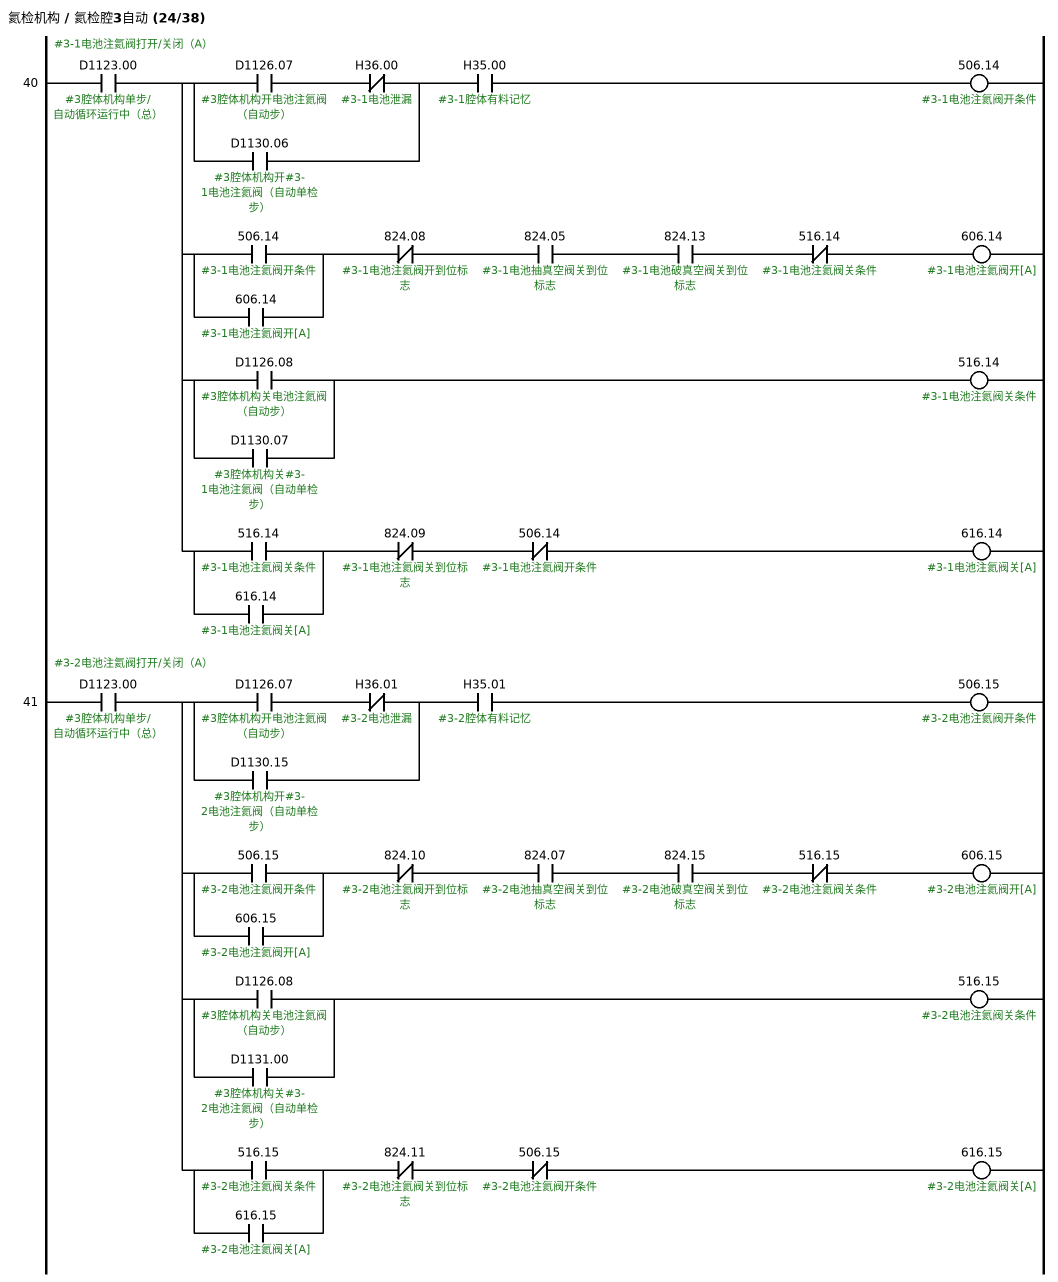
; [picture p312: 氦检机构 / 氦检腔3自动, rungs 40-41]
; rung 40: #3-1电池注氦阀打开/关闭（A）
LD D1123.00  ; #3腔体机构单步/自动循环运行中（总）
OUT TR0
LD D1126.07  ; #3腔体机构开电池注氦阀（自动步）
ANDNOT H36.00  ; #3-1电池泄漏
OR D1130.06  ; #3腔体机构开#3-1电池注氦阀（自动单检步）
ANDLD
AND H35.00  ; #3-1腔体有料记忆
OUT 506.14  ; #3-1电池注氦阀开条件
LD TR0
LD 506.14  ; #3-1电池注氦阀开条件
OR 606.14  ; #3-1电池注氦阀开[A]
ANDLD
ANDNOT 824.08  ; #3-1电池注氦阀开到位标志
AND 824.05  ; #3-1电池抽真空阀关到位标志
AND 824.13  ; #3-1电池破真空阀关到位标志
ANDNOT 516.14  ; #3-1电池注氦阀关条件
OUT 606.14  ; #3-1电池注氦阀开[A]
LD TR0
LD D1126.08  ; #3腔体机构关电池注氦阀（自动步）
OR D1130.07  ; #3腔体机构关#3-1电池注氦阀（自动单检步）
ANDLD
OUT 516.14  ; #3-1电池注氦阀关条件
LD TR0
LD 516.14  ; #3-1电池注氦阀关条件
OR 616.14  ; #3-1电池注氦阀关[A]
ANDLD
ANDNOT 824.09  ; #3-1电池注氦阀关到位标志
ANDNOT 506.14  ; #3-1电池注氦阀开条件
OUT 616.14  ; #3-1电池注氦阀关[A]
; rung 41: #3-2电池注氦阀打开/关闭（A）
LD D1123.00  ; #3腔体机构单步/自动循环运行中（总）
OUT TR0
LD D1126.07  ; #3腔体机构开电池注氦阀（自动步）
ANDNOT H36.01  ; #3-2电池泄漏
OR D1130.15  ; #3腔体机构开#3-2电池注氦阀（自动单检步）
ANDLD
AND H35.01  ; #3-2腔体有料记忆
OUT 506.15  ; #3-2电池注氦阀开条件
LD TR0
LD 506.15  ; #3-2电池注氦阀开条件
OR 606.15  ; #3-2电池注氦阀开[A]
ANDLD
ANDNOT 824.10  ; #3-2电池注氦阀开到位标志
AND 824.07  ; #3-2电池抽真空阀关到位标志
AND 824.15  ; #3-2电池破真空阀关到位标志
ANDNOT 516.15  ; #3-2电池注氦阀关条件
OUT 606.15  ; #3-2电池注氦阀开[A]
LD TR0
LD D1126.08  ; #3腔体机构关电池注氦阀（自动步）
OR D1131.00  ; #3腔体机构关#3-2电池注氦阀（自动单检步）
ANDLD
OUT 516.15  ; #3-2电池注氦阀关条件
LD TR0
LD 516.15  ; #3-2电池注氦阀关条件
OR 616.15  ; #3-2电池注氦阀关[A]
ANDLD
ANDNOT 824.11  ; #3-2电池注氦阀关到位标志
ANDNOT 506.15  ; #3-2电池注氦阀开条件
OUT 616.15  ; #3-2电池注氦阀关[A]

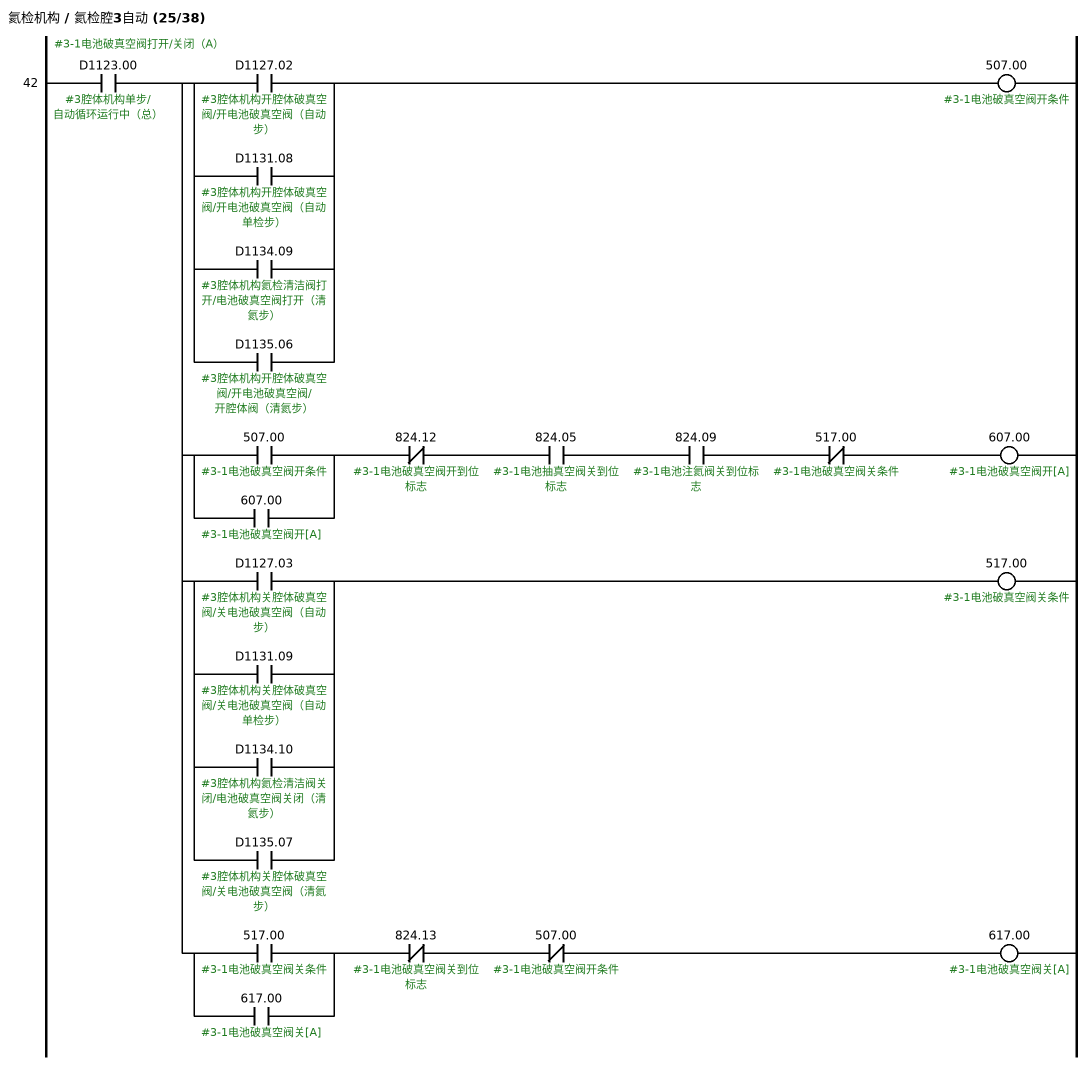
; rung 42: #3-1电池破真空阀打开/关闭（A）
LD D1123.00  ; #3腔体机构单步/自动循环运行中（总）
OUT TR0
LD D1127.02  ; #3腔体机构开腔体破真空阀/开电池破真空阀（自动步）
OR D1131.08  ; #3腔体机构开腔体破真空阀/开电池破真空阀（自动单检步）
OR D1134.09  ; #3腔体机构氦检清洁阀打开/电池破真空阀打开（清氦步）
OR D1135.06  ; #3腔体机构开腔体破真空阀/开电池破真空阀/开腔体阀（清氦步）
ANDLD
OUT 507.00  ; #3-1电池破真空阀开条件
LD TR0
LD 507.00  ; #3-1电池破真空阀开条件
OR 607.00  ; #3-1电池破真空阀开[A]
ANDLD
ANDNOT 824.12  ; #3-1电池破真空阀开到位标志
AND 824.05  ; #3-1电池抽真空阀关到位标志
AND 824.09  ; #3-1电池注氦阀关到位标志
ANDNOT 517.00  ; #3-1电池破真空阀关条件
OUT 607.00  ; #3-1电池破真空阀开[A]
LD TR0
LD D1127.03  ; #3腔体机构关腔体破真空阀/关电池破真空阀（自动步）
OR D1131.09  ; #3腔体机构关腔体破真空阀/关电池破真空阀（自动单检步）
OR D1134.10  ; #3腔体机构氦检清洁阀关闭/电池破真空阀关闭（清氦步）
OR D1135.07  ; #3腔体机构关腔体破真空阀/关电池破真空阀（清氦步）
ANDLD
OUT 517.00  ; #3-1电池破真空阀关条件
LD TR0
LD 517.00  ; #3-1电池破真空阀关条件
OR 617.00  ; #3-1电池破真空阀关[A]
ANDLD
ANDNOT 824.13  ; #3-1电池破真空阀关到位标志
ANDNOT 507.00  ; #3-1电池破真空阀开条件
OUT 617.00  ; #3-1电池破真空阀关[A]

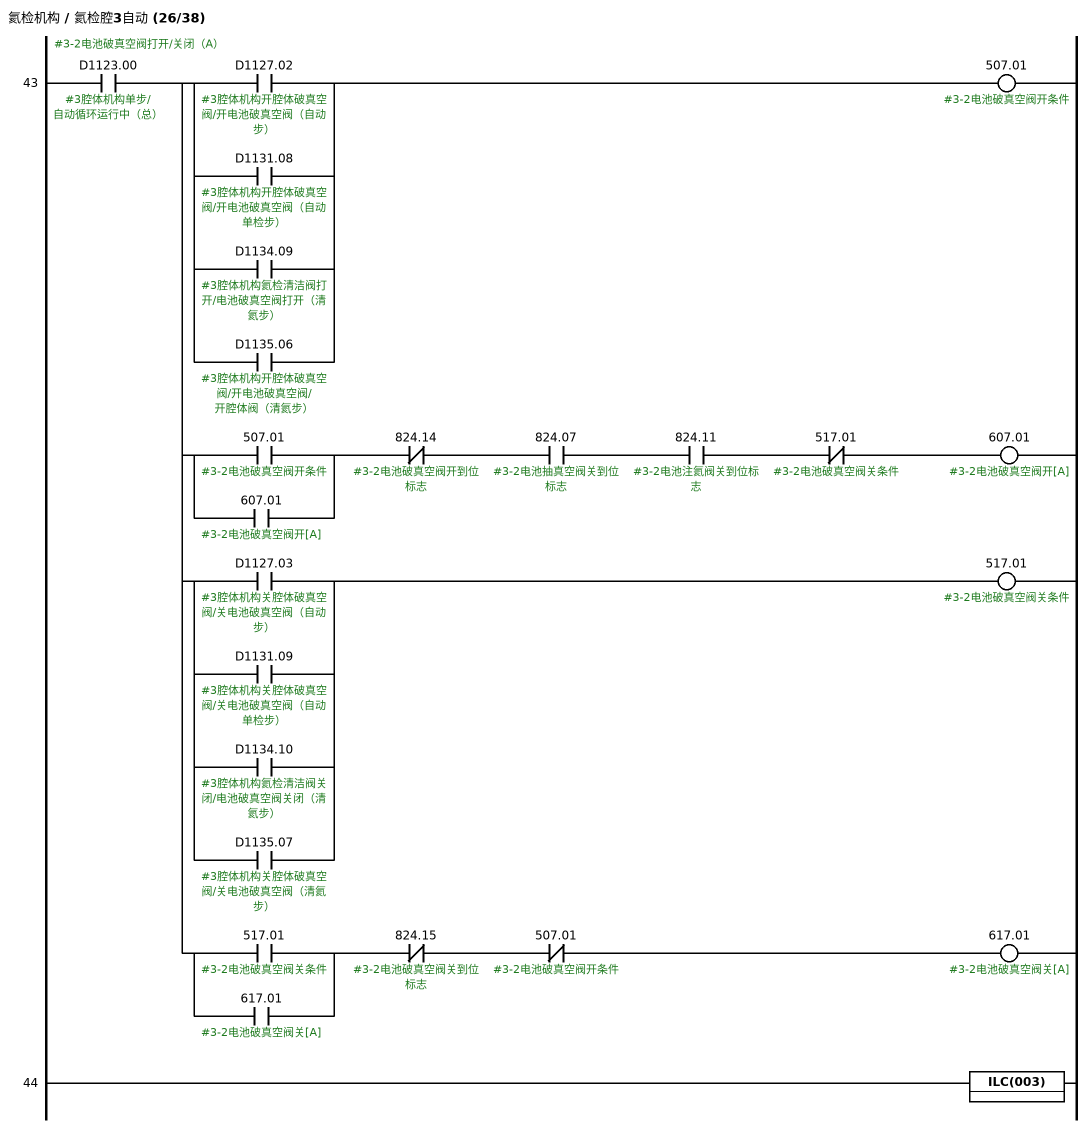
; rung 43: #3-2电池破真空阀打开/关闭（A）
LD D1123.00  ; #3腔体机构单步/自动循环运行中（总）
OUT TR0
LD D1127.02  ; #3腔体机构开腔体破真空阀/开电池破真空阀（自动步）
OR D1131.08  ; #3腔体机构开腔体破真空阀/开电池破真空阀（自动单检步）
OR D1134.09  ; #3腔体机构氦检清洁阀打开/电池破真空阀打开（清氦步）
OR D1135.06  ; #3腔体机构开腔体破真空阀/开电池破真空阀/开腔体阀（清氦步）
ANDLD
OUT 507.01  ; #3-2电池破真空阀开条件
LD TR0
LD 507.01  ; #3-2电池破真空阀开条件
OR 607.01  ; #3-2电池破真空阀开[A]
ANDLD
ANDNOT 824.14  ; #3-2电池破真空阀开到位标志
AND 824.07  ; #3-2电池抽真空阀关到位标志
AND 824.11  ; #3-2电池注氦阀关到位标志
ANDNOT 517.01  ; #3-2电池破真空阀关条件
OUT 607.01  ; #3-2电池破真空阀开[A]
LD TR0
LD D1127.03  ; #3腔体机构关腔体破真空阀/关电池破真空阀（自动步）
OR D1131.09  ; #3腔体机构关腔体破真空阀/关电池破真空阀（自动单检步）
OR D1134.10  ; #3腔体机构氦检清洁阀关闭/电池破真空阀关闭（清氦步）
OR D1135.07  ; #3腔体机构关腔体破真空阀/关电池破真空阀（清氦步）
ANDLD
OUT 517.01  ; #3-2电池破真空阀关条件
LD TR0
LD 517.01  ; #3-2电池破真空阀关条件
OR 617.01  ; #3-2电池破真空阀关[A]
ANDLD
ANDNOT 824.15  ; #3-2电池破真空阀关到位标志
ANDNOT 507.01  ; #3-2电池破真空阀开条件
OUT 617.01  ; #3-2电池破真空阀关[A]
; rung 44
ILC(003)

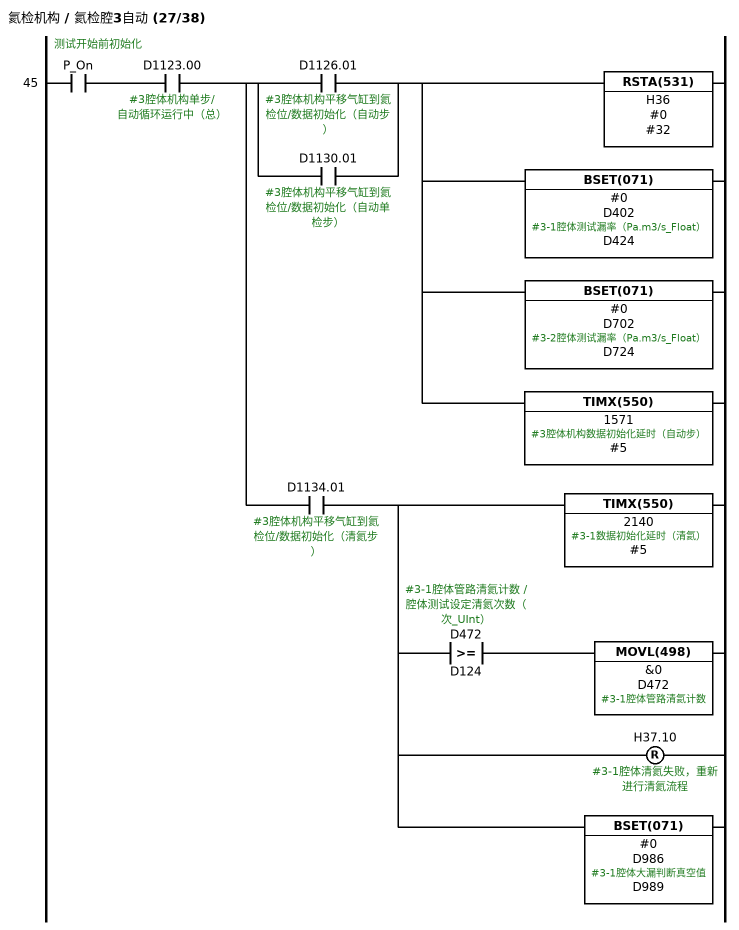
; rung 45: 测试开始前初始化
LD P_On
AND D1123.00  ; #3腔体机构单步/自动循环运行中（总）
OUT TR0
LD D1126.01  ; #3腔体机构平移气缸到氦检位/数据初始化（自动步）
OR D1130.01  ; #3腔体机构平移气缸到氦检位/数据初始化（自动单检步）
ANDLD
RSTA(531) H36 #0 #32
BSET(071) #0 D402 D424  ; #3-1腔体测试漏率（Pa.m3/s_Float）
BSET(071) #0 D702 D724  ; #3-2腔体测试漏率（Pa.m3/s_Float）
TIMX(550) 1571 #5  ; #3腔体机构数据初始化延时（自动步）
LD TR0
AND D1134.01  ; #3腔体机构平移气缸到氦检位/数据初始化（清氦步）
OUT TR0
TIMX(550) 2140 #5  ; #3-1数据初始化延时（清氦）
AND>=(325) D472 D124  ; #3-1腔体管路清氦计数, 腔体测试设定清氦次数（次_UInt）
MOVL(498) &0 D472  ; #3-1腔体管路清氦计数
LD TR0
RSET H37.10  ; #3-1腔体清氦失败，重新进行清氦流程
BSET(071) #0 D986 D989  ; #3-1腔体大漏判断真空值

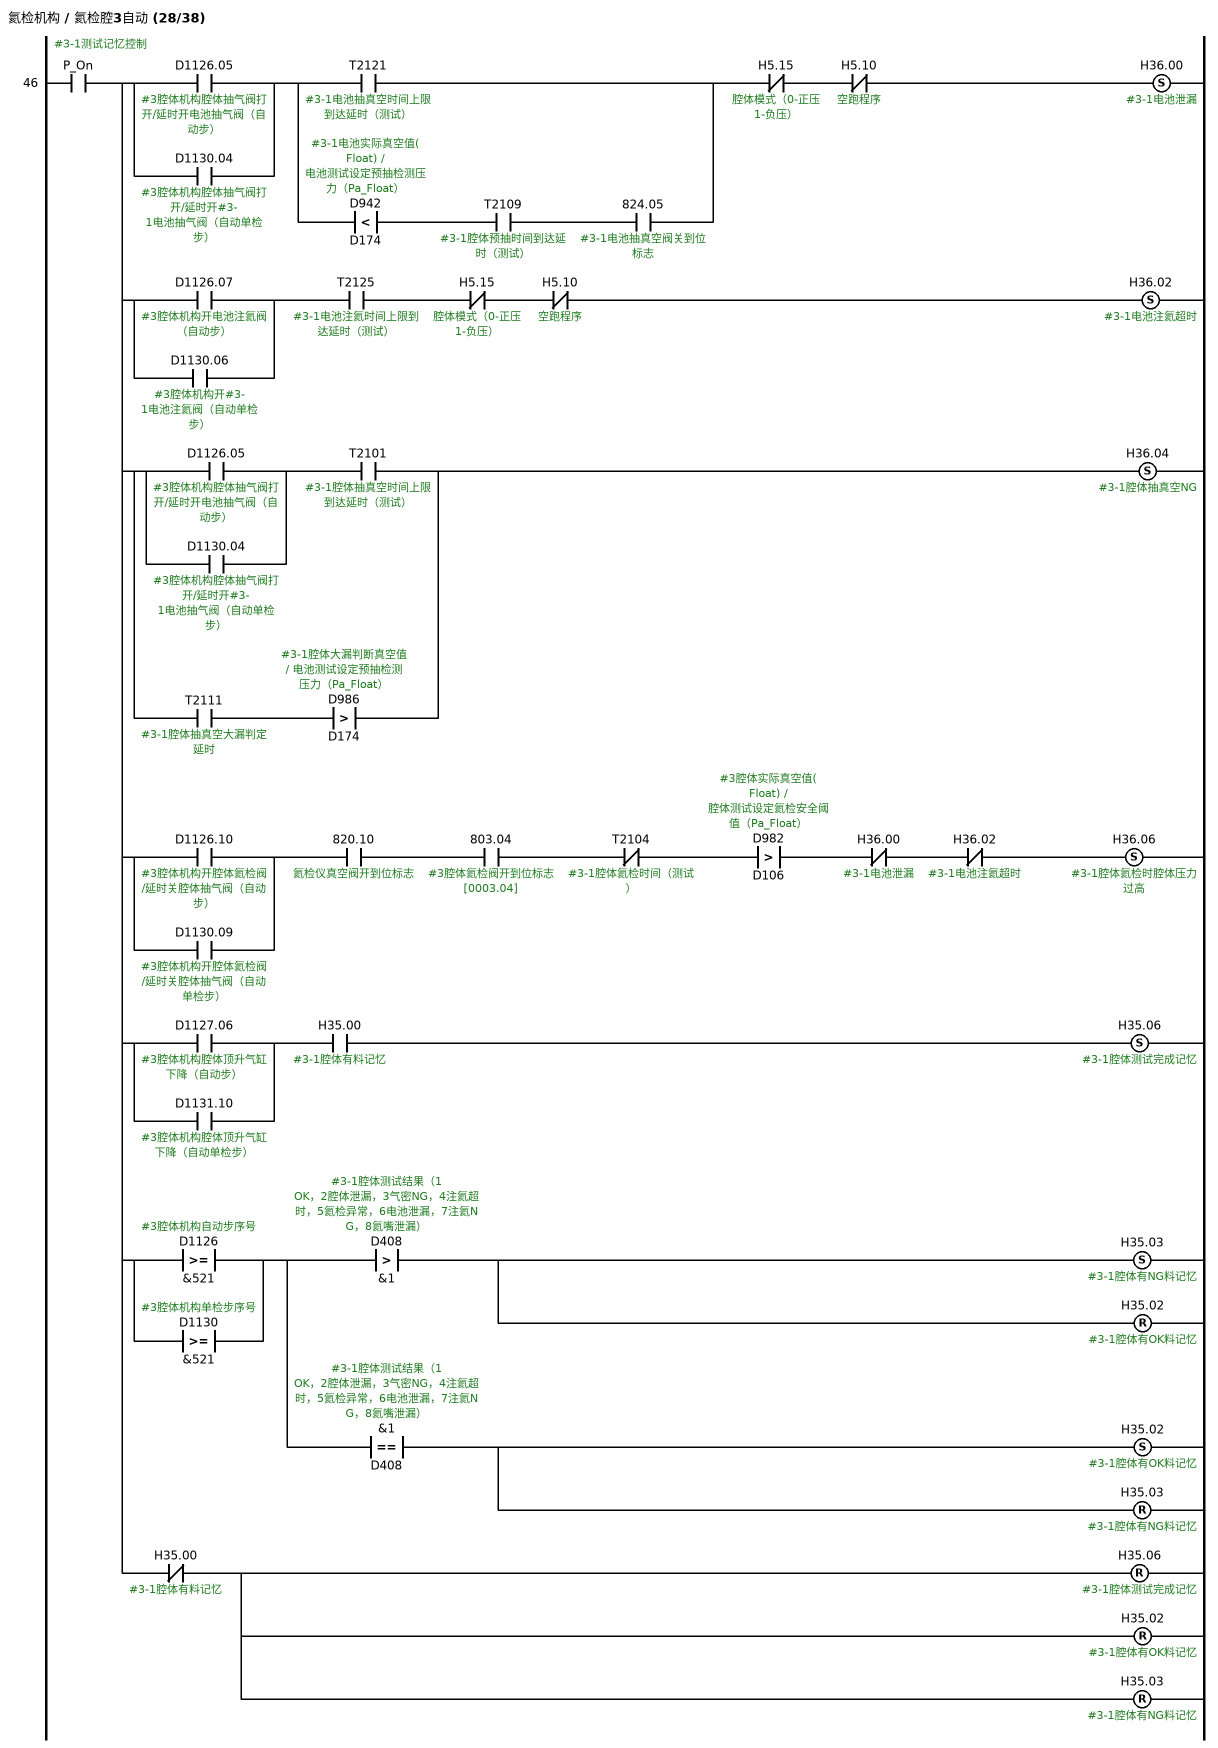
; rung 46: #3-1测试记忆控制
LD P_On
OUT TR0
LD D1126.05  ; #3腔体机构腔体抽气阀打开/延时开电池抽气阀（自动步）
OR D1130.04  ; #3腔体机构腔体抽气阀打开/延时开#3-1电池抽气阀（自动单检步）
ANDLD
LD T2121  ; #3-1电池抽真空时间上限到达延时（测试）
LD<F(331) D942 D174  ; #3-1电池实际真空值(Float), 电池测试设定预抽检测压力（Pa_Float）
AND T2109  ; #3-1腔体预抽时间到达延时（测试）
AND 824.05  ; #3-1电池抽真空阀关到位标志
ORLD
ANDLD
ANDNOT H5.15  ; 腔体模式（0-正压 1-负压）
ANDNOT H5.10  ; 空跑程序
SET H36.00  ; #3-1电池泄漏
LD TR0
LD D1126.07  ; #3腔体机构开电池注氦阀（自动步）
OR D1130.06  ; #3腔体机构开#3-1电池注氦阀（自动单检步）
ANDLD
AND T2125  ; #3-1电池注氦时间上限到达延时（测试）
ANDNOT H5.15  ; 腔体模式（0-正压 1-负压）
ANDNOT H5.10  ; 空跑程序
SET H36.02  ; #3-1电池注氦超时
LD TR0
LD D1126.05  ; #3腔体机构腔体抽气阀打开/延时开电池抽气阀（自动步）
OR D1130.04  ; #3腔体机构腔体抽气阀打开/延时开#3-1电池抽气阀（自动单检步）
AND T2101  ; #3-1腔体抽真空时间上限到达延时（测试）
LD T2111  ; #3-1腔体抽真空大漏判定延时
AND>F(333) D986 D174  ; #3-1腔体大漏判断真空值, 电池测试设定预抽检测压力（Pa_Float）
ORLD
ANDLD
SET H36.04  ; #3-1腔体抽真空NG
LD TR0
LD D1126.10  ; #3腔体机构开腔体氦检阀/延时关腔体抽气阀（自动步）
OR D1130.09  ; #3腔体机构开腔体氦检阀/延时关腔体抽气阀（自动单检步）
ANDLD
AND 820.10  ; 氦检仪真空阀开到位标志
AND 803.04  ; #3腔体氦检阀开到位标志[0003.04]
ANDNOT T2104  ; #3-1腔体氦检时间（测试）
AND>F(333) D982 D106  ; #3腔体实际真空值(Float), 腔体测试设定氦检安全阈值（Pa_Float）
ANDNOT H36.00  ; #3-1电池泄漏
ANDNOT H36.02  ; #3-1电池注氦超时
SET H36.06  ; #3-1腔体氦检时腔体压力过高
LD TR0
LD D1127.06  ; #3腔体机构腔体顶升气缸下降（自动步）
OR D1131.10  ; #3腔体机构腔体顶升气缸下降（自动单检步）
ANDLD
AND H35.00  ; #3-1腔体有料记忆
SET H35.06  ; #3-1腔体测试完成记忆
LD TR0
LD>=L(326) D1126 &521  ; #3腔体机构自动步序号
OR>=L(326) D1130 &521  ; #3腔体机构单检步序号
ANDLD
OUT TR1
AND>(320) D408 &1  ; #3-1腔体测试结果（1 OK，2腔体泄漏，3气密NG，4注氦超时，5氦检异常，6电池泄漏，7注氦NG，8氦嘴泄漏）
SET H35.03  ; #3-1腔体有NG料记忆
RSET H35.02  ; #3-1腔体有OK料记忆
LD TR1
AND=(300) &1 D408  ; #3-1腔体测试结果（1 OK，2腔体泄漏，3气密NG，4注氦超时，5氦检异常，6电池泄漏，7注氦NG，8氦嘴泄漏）
SET H35.02  ; #3-1腔体有OK料记忆
RSET H35.03  ; #3-1腔体有NG料记忆
LD TR0
ANDNOT H35.00  ; #3-1腔体有料记忆
RSET H35.06  ; #3-1腔体测试完成记忆
RSET H35.02  ; #3-1腔体有OK料记忆
RSET H35.03  ; #3-1腔体有NG料记忆

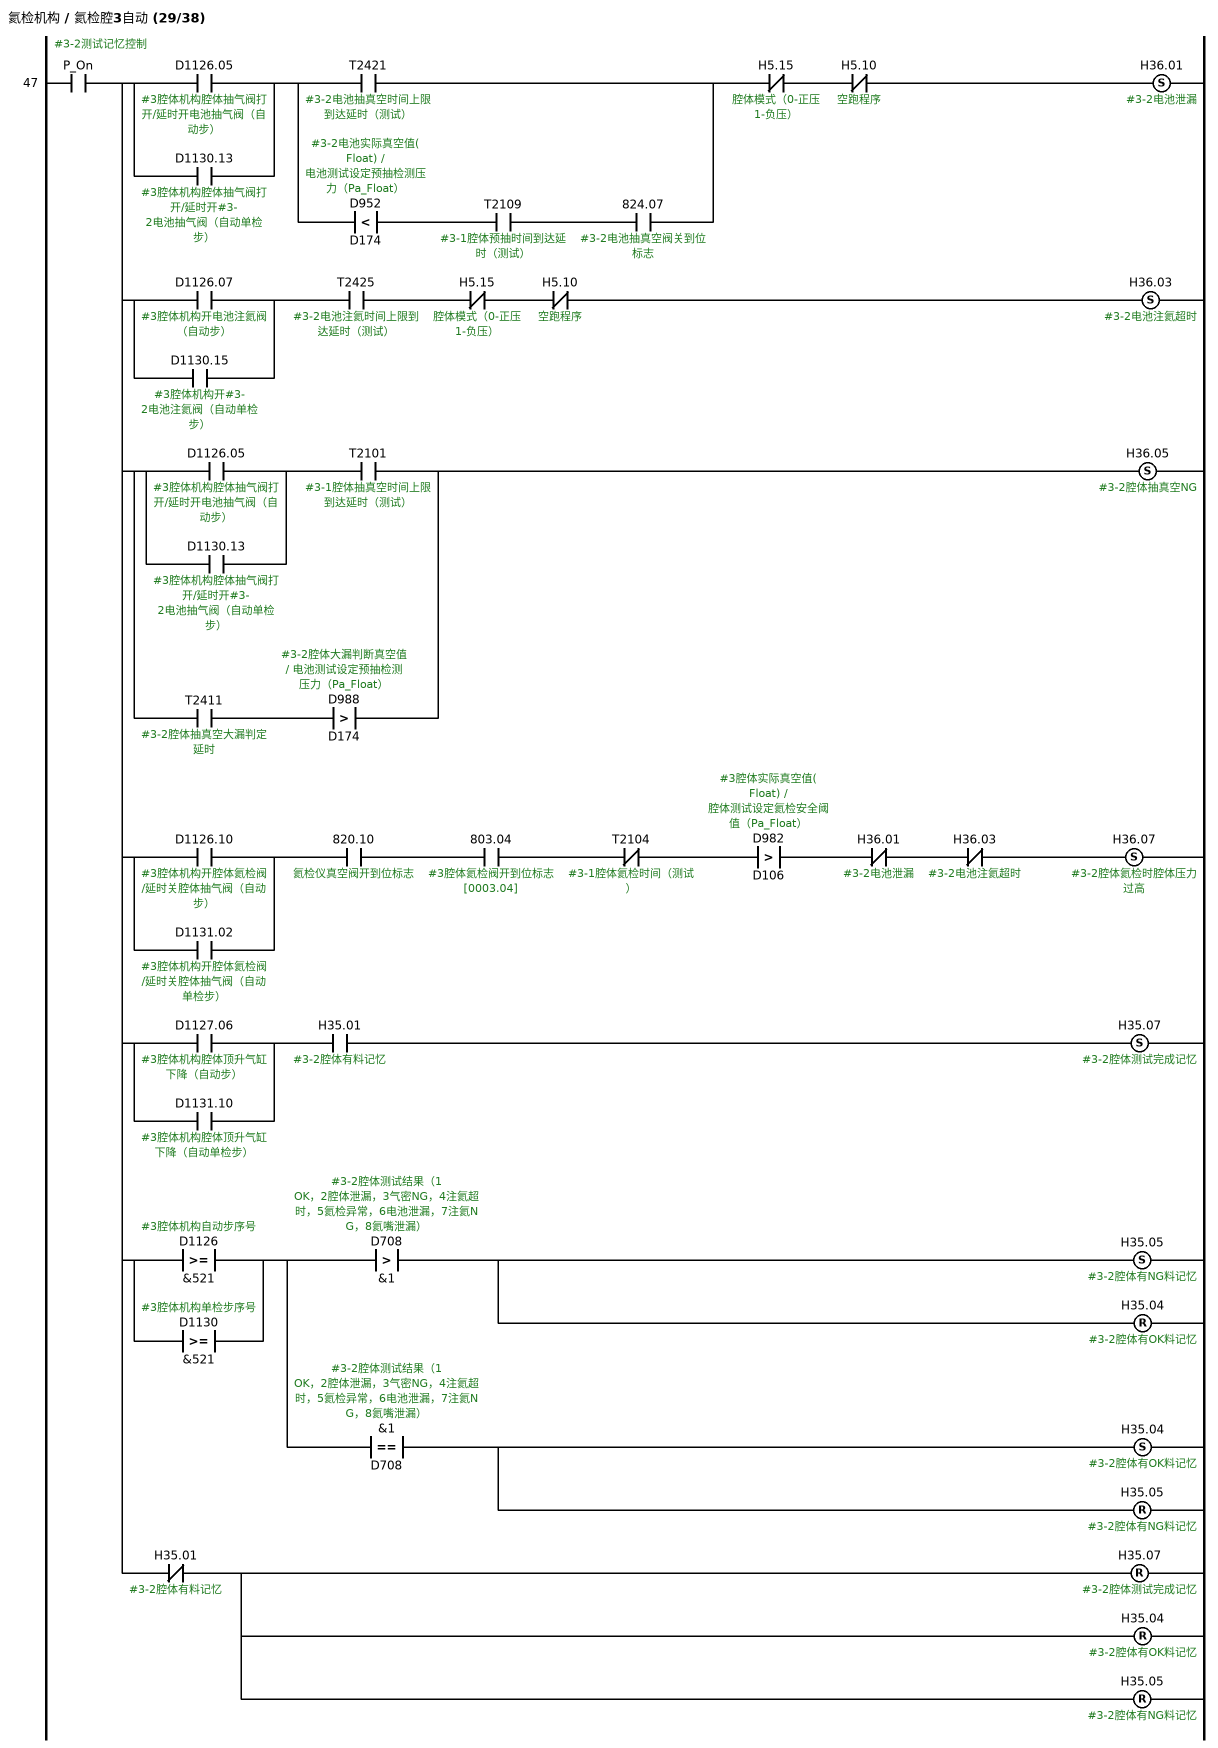
; rung 47: #3-2测试记忆控制
LD P_On
OUT TR0
LD D1126.05  ; #3腔体机构腔体抽气阀打开/延时开电池抽气阀（自动步）
OR D1130.13  ; #3腔体机构腔体抽气阀打开/延时开#3-2电池抽气阀（自动单检步）
ANDLD
LD T2421  ; #3-2电池抽真空时间上限到达延时（测试）
LD<F(331) D952 D174  ; #3-2电池实际真空值(Float), 电池测试设定预抽检测压力（Pa_Float）
AND T2109  ; #3-1腔体预抽时间到达延时（测试）
AND 824.07  ; #3-2电池抽真空阀关到位标志
ORLD
ANDLD
ANDNOT H5.15  ; 腔体模式（0-正压 1-负压）
ANDNOT H5.10  ; 空跑程序
SET H36.01  ; #3-2电池泄漏
LD TR0
LD D1126.07  ; #3腔体机构开电池注氦阀（自动步）
OR D1130.15  ; #3腔体机构开#3-2电池注氦阀（自动单检步）
ANDLD
AND T2425  ; #3-2电池注氦时间上限到达延时（测试）
ANDNOT H5.15  ; 腔体模式（0-正压 1-负压）
ANDNOT H5.10  ; 空跑程序
SET H36.03  ; #3-2电池注氦超时
LD TR0
LD D1126.05  ; #3腔体机构腔体抽气阀打开/延时开电池抽气阀（自动步）
OR D1130.13  ; #3腔体机构腔体抽气阀打开/延时开#3-2电池抽气阀（自动单检步）
AND T2101  ; #3-1腔体抽真空时间上限到达延时（测试）
LD T2411  ; #3-2腔体抽真空大漏判定延时
AND>F(333) D988 D174  ; #3-2腔体大漏判断真空值, 电池测试设定预抽检测压力（Pa_Float）
ORLD
ANDLD
SET H36.05  ; #3-2腔体抽真空NG
LD TR0
LD D1126.10  ; #3腔体机构开腔体氦检阀/延时关腔体抽气阀（自动步）
OR D1131.02  ; #3腔体机构开腔体氦检阀/延时关腔体抽气阀（自动单检步）
ANDLD
AND 820.10  ; 氦检仪真空阀开到位标志
AND 803.04  ; #3腔体氦检阀开到位标志[0003.04]
ANDNOT T2104  ; #3-1腔体氦检时间（测试）
AND>F(333) D982 D106  ; #3腔体实际真空值(Float), 腔体测试设定氦检安全阈值（Pa_Float）
ANDNOT H36.01  ; #3-2电池泄漏
ANDNOT H36.03  ; #3-2电池注氦超时
SET H36.07  ; #3-2腔体氦检时腔体压力过高
LD TR0
LD D1127.06  ; #3腔体机构腔体顶升气缸下降（自动步）
OR D1131.10  ; #3腔体机构腔体顶升气缸下降（自动单检步）
ANDLD
AND H35.01  ; #3-2腔体有料记忆
SET H35.07  ; #3-2腔体测试完成记忆
LD TR0
LD>=L(326) D1126 &521  ; #3腔体机构自动步序号
OR>=L(326) D1130 &521  ; #3腔体机构单检步序号
ANDLD
OUT TR1
AND>(320) D708 &1  ; #3-2腔体测试结果（1 OK，2腔体泄漏，3气密NG，4注氦超时，5氦检异常，6电池泄漏，7注氦NG，8氦嘴泄漏）
SET H35.05  ; #3-2腔体有NG料记忆
RSET H35.04  ; #3-2腔体有OK料记忆
LD TR1
AND=(300) &1 D708  ; #3-2腔体测试结果（1 OK，2腔体泄漏，3气密NG，4注氦超时，5氦检异常，6电池泄漏，7注氦NG，8氦嘴泄漏）
SET H35.04  ; #3-2腔体有OK料记忆
RSET H35.05  ; #3-2腔体有NG料记忆
LD TR0
ANDNOT H35.01  ; #3-2腔体有料记忆
RSET H35.07  ; #3-2腔体测试完成记忆
RSET H35.04  ; #3-2腔体有OK料记忆
RSET H35.05  ; #3-2腔体有NG料记忆

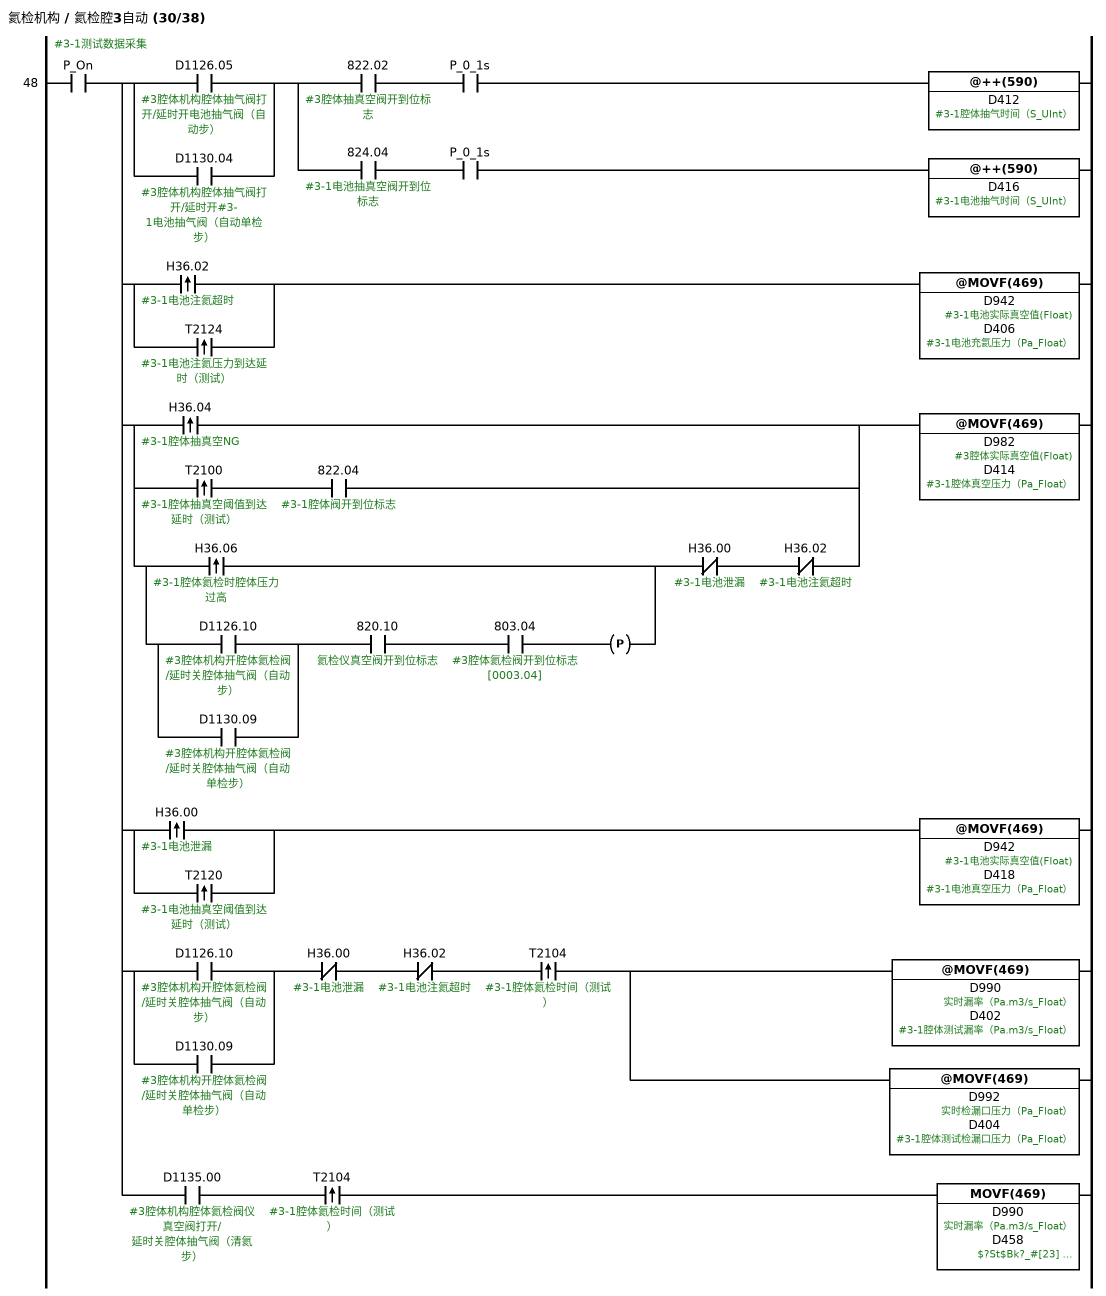
; rung 48: #3-1测试数据采集
LD P_On
OUT TR0
LD D1126.05  ; #3腔体机构腔体抽气阀打开/延时开电池抽气阀（自动步）
OR D1130.04  ; #3腔体机构腔体抽气阀打开/延时开#3-1电池抽气阀（自动单检步）
ANDLD
OUT TR1
AND 822.02  ; #3腔体抽真空阀开到位标志
AND P_0_1s
@++(590) D412  ; #3-1腔体抽气时间（S_UInt）
LD TR1
AND 824.04  ; #3-1电池抽真空阀开到位标志
AND P_0_1s
@++(590) D416  ; #3-1电池抽气时间（S_UInt）
LD TR0
@LD H36.02  ; #3-1电池注氦超时
@OR T2124  ; #3-1电池注氦压力到达延时（测试）
ANDLD
@MOVF(469) D942 D406  ; #3-1电池实际真空值(Float), #3-1电池充氦压力（Pa_Float）
LD TR0
@LD H36.04  ; #3-1腔体抽真空NG
@LD T2100  ; #3-1腔体抽真空阈值到达延时（测试）
AND 822.04  ; #3-1腔体阀开到位标志
ORLD
@LD H36.06  ; #3-1腔体氦检时腔体压力过高
LD D1126.10  ; #3腔体机构开腔体氦检阀/延时关腔体抽气阀（自动步）
OR D1130.09  ; #3腔体机构开腔体氦检阀/延时关腔体抽气阀（自动单检步）
AND 820.10  ; 氦检仪真空阀开到位标志
AND 803.04  ; #3腔体氦检阀开到位标志[0003.04]
UP(521)
ORLD
ANDNOT H36.00  ; #3-1电池泄漏
ANDNOT H36.02  ; #3-1电池注氦超时
ORLD
ANDLD
@MOVF(469) D982 D414  ; #3腔体实际真空值(Float), #3-1腔体真空压力（Pa_Float）
LD TR0
@LD H36.00  ; #3-1电池泄漏
@OR T2120  ; #3-1电池抽真空阈值到达延时（测试）
ANDLD
@MOVF(469) D942 D418  ; #3-1电池实际真空值(Float), #3-1电池真空压力（Pa_Float）
LD TR0
LD D1126.10  ; #3腔体机构开腔体氦检阀/延时关腔体抽气阀（自动步）
OR D1130.09  ; #3腔体机构开腔体氦检阀/延时关腔体抽气阀（自动单检步）
ANDLD
ANDNOT H36.00  ; #3-1电池泄漏
ANDNOT H36.02  ; #3-1电池注氦超时
@AND T2104  ; #3-1腔体氦检时间（测试）
@MOVF(469) D990 D402  ; 实时漏率（Pa.m3/s_Float）, #3-1腔体测试漏率（Pa.m3/s_Float）
@MOVF(469) D992 D404  ; 实时检漏口压力（Pa_Float）, #3-1腔体测试检漏口压力（Pa_Float）
LD TR0
AND D1135.00  ; #3腔体机构腔体氦检阀仪真空阀打开/延时关腔体抽气阀（清氦步）
@AND T2104  ; #3-1腔体氦检时间（测试）
MOVF(469) D990 D458  ; 实时漏率（Pa.m3/s_Float）, $?St$Bk?_#[23] / #3-1清氦泄漏率（清氦） / $?St$Bk?_#[23]

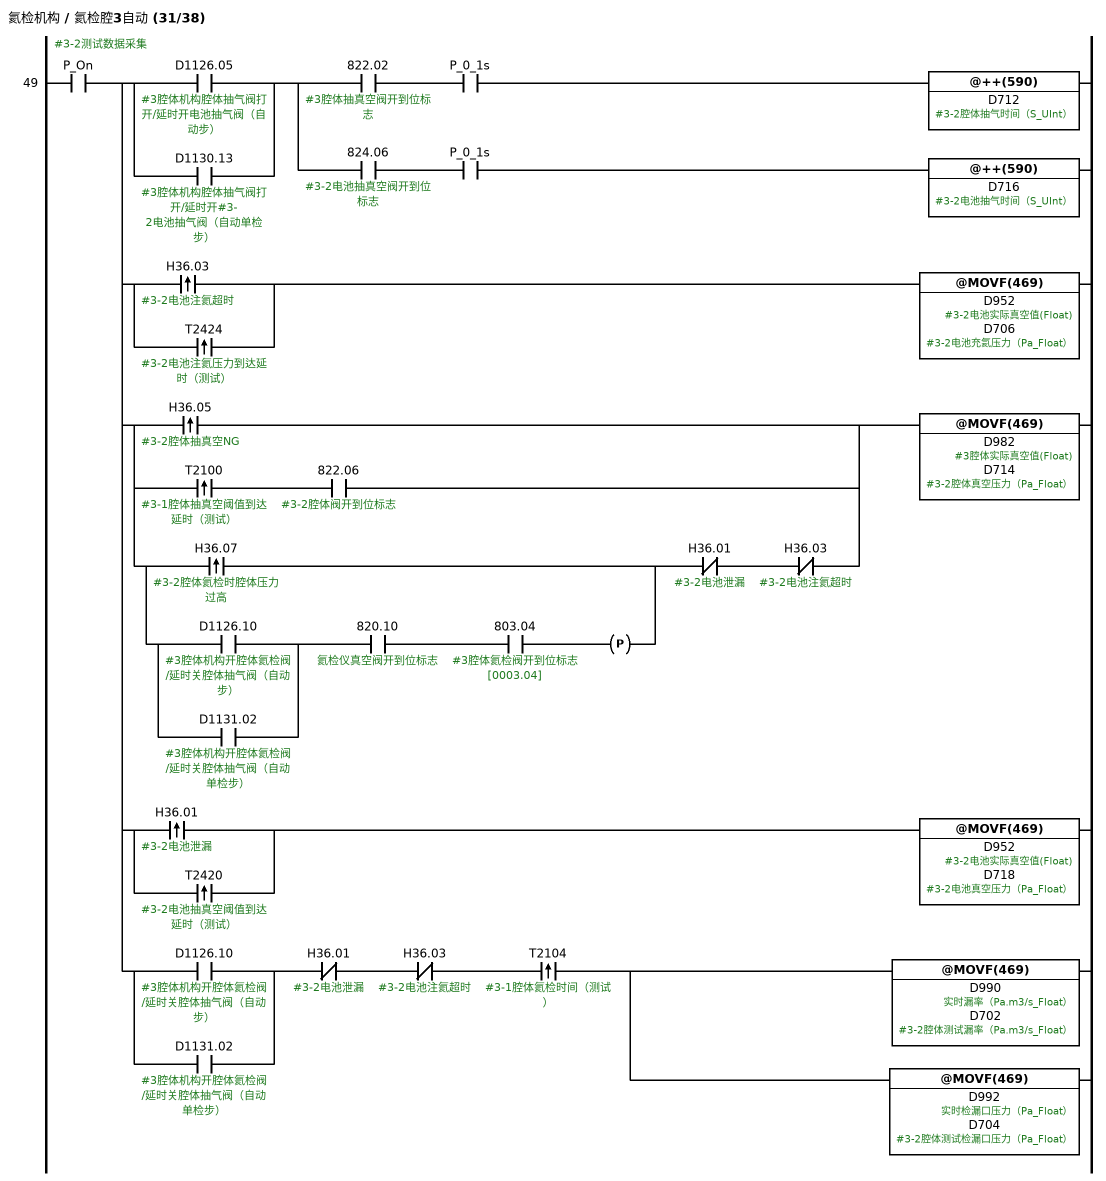
; rung 49: #3-2测试数据采集
LD P_On
OUT TR0
LD D1126.05  ; #3腔体机构腔体抽气阀打开/延时开电池抽气阀（自动步）
OR D1130.13  ; #3腔体机构腔体抽气阀打开/延时开#3-2电池抽气阀（自动单检步）
ANDLD
OUT TR1
AND 822.02  ; #3腔体抽真空阀开到位标志
AND P_0_1s
@++(590) D712  ; #3-2腔体抽气时间（S_UInt）
LD TR1
AND 824.06  ; #3-2电池抽真空阀开到位标志
AND P_0_1s
@++(590) D716  ; #3-2电池抽气时间（S_UInt）
LD TR0
@LD H36.03  ; #3-2电池注氦超时
@OR T2424  ; #3-2电池注氦压力到达延时（测试）
ANDLD
@MOVF(469) D952 D706  ; #3-2电池实际真空值(Float), #3-2电池充氦压力（Pa_Float）
LD TR0
@LD H36.05  ; #3-2腔体抽真空NG
@LD T2100  ; #3-1腔体抽真空阈值到达延时（测试）
AND 822.06  ; #3-2腔体阀开到位标志
ORLD
@LD H36.07  ; #3-2腔体氦检时腔体压力过高
LD D1126.10  ; #3腔体机构开腔体氦检阀/延时关腔体抽气阀（自动步）
OR D1131.02  ; #3腔体机构开腔体氦检阀/延时关腔体抽气阀（自动单检步）
AND 820.10  ; 氦检仪真空阀开到位标志
AND 803.04  ; #3腔体氦检阀开到位标志[0003.04]
UP(521)
ORLD
ANDNOT H36.01  ; #3-2电池泄漏
ANDNOT H36.03  ; #3-2电池注氦超时
ORLD
ANDLD
@MOVF(469) D982 D714  ; #3腔体实际真空值(Float), #3-2腔体真空压力（Pa_Float）
LD TR0
@LD H36.01  ; #3-2电池泄漏
@OR T2420  ; #3-2电池抽真空阈值到达延时（测试）
ANDLD
@MOVF(469) D952 D718  ; #3-2电池实际真空值(Float), #3-2电池真空压力（Pa_Float）
LD TR0
LD D1126.10  ; #3腔体机构开腔体氦检阀/延时关腔体抽气阀（自动步）
OR D1131.02  ; #3腔体机构开腔体氦检阀/延时关腔体抽气阀（自动单检步）
ANDLD
ANDNOT H36.01  ; #3-2电池泄漏
ANDNOT H36.03  ; #3-2电池注氦超时
@AND T2104  ; #3-1腔体氦检时间（测试）
@MOVF(469) D990 D702  ; 实时漏率（Pa.m3/s_Float）, #3-2腔体测试漏率（Pa.m3/s_Float）
@MOVF(469) D992 D704  ; 实时检漏口压力（Pa_Float）, #3-2腔体测试检漏口压力（Pa_Float）

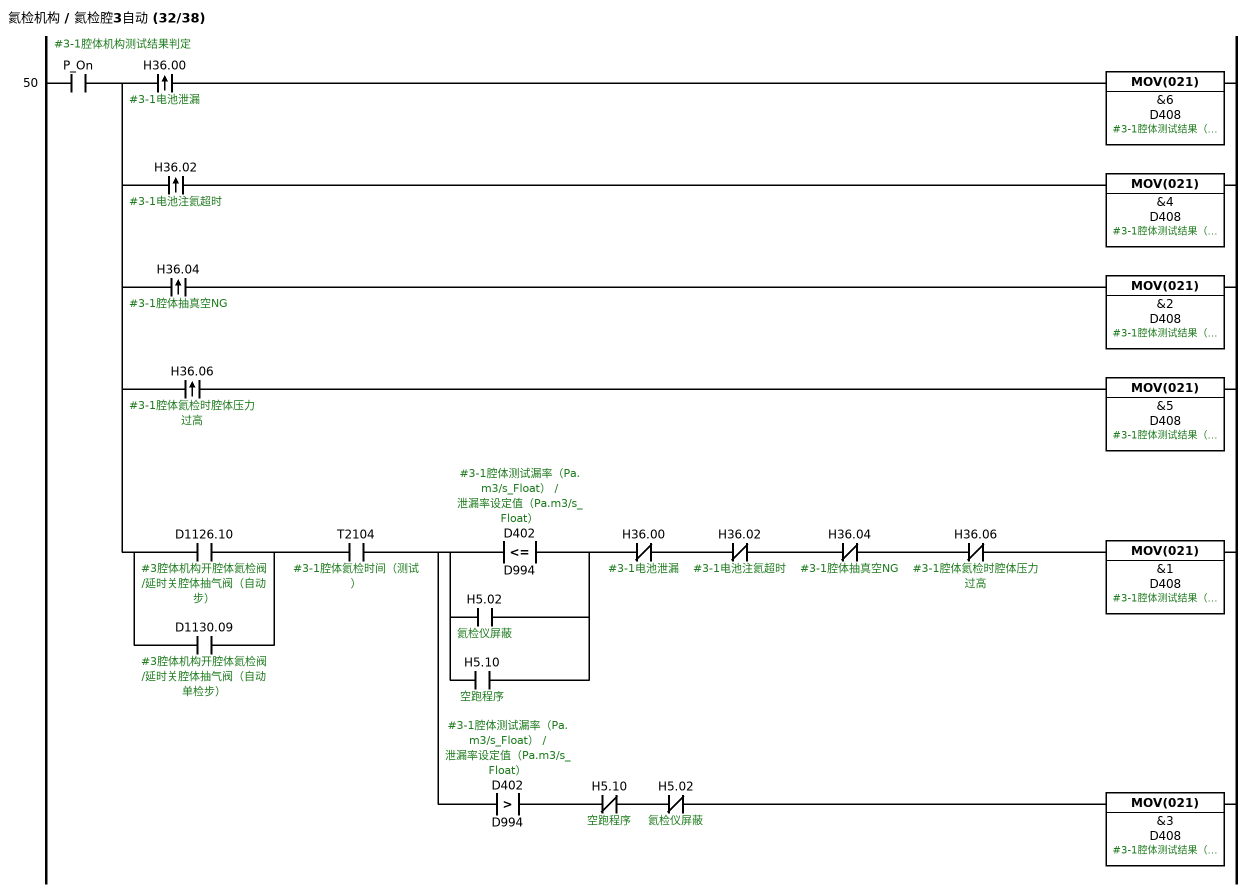
; rung 50: #3-1腔体机构测试结果判定
LD P_On
OUT TR0
@AND H36.00  ; #3-1电池泄漏
MOV(021) &6 D408  ; #3-1腔体测试结果（1 OK，2腔体泄漏，3气密NG，4注氦超时，5氦检异常，6电池泄漏，7注氦NG，8氦嘴泄漏）
LD TR0
@AND H36.02  ; #3-1电池注氦超时
MOV(021) &4 D408  ; #3-1腔体测试结果（1 OK，2腔体泄漏，3气密NG，4注氦超时，5氦检异常，6电池泄漏，7注氦NG，8氦嘴泄漏）
LD TR0
@AND H36.04  ; #3-1腔体抽真空NG
MOV(021) &2 D408  ; #3-1腔体测试结果（1 OK，2腔体泄漏，3气密NG，4注氦超时，5氦检异常，6电池泄漏，7注氦NG，8氦嘴泄漏）
LD TR0
@AND H36.06  ; #3-1腔体氦检时腔体压力过高
MOV(021) &5 D408  ; #3-1腔体测试结果（1 OK，2腔体泄漏，3气密NG，4注氦超时，5氦检异常，6电池泄漏，7注氦NG，8氦嘴泄漏）
LD TR0
LD D1126.10  ; #3腔体机构开腔体氦检阀/延时关腔体抽气阀（自动步）
OR D1130.09  ; #3腔体机构开腔体氦检阀/延时关腔体抽气阀（自动单检步）
ANDLD
AND T2104  ; #3-1腔体氦检时间（测试）
OUT TR0
LD<=F(332) D402 D994  ; #3-1腔体测试漏率（Pa.m3/s_Float）, 泄漏率设定值（Pa.m3/s_Float）
OR H5.02  ; 氦检仪屏蔽
OR H5.10  ; 空跑程序
ANDLD
ANDNOT H36.00  ; #3-1电池泄漏
ANDNOT H36.02  ; #3-1电池注氦超时
ANDNOT H36.04  ; #3-1腔体抽真空NG
ANDNOT H36.06  ; #3-1腔体氦检时腔体压力过高
MOV(021) &1 D408  ; #3-1腔体测试结果（1 OK，2腔体泄漏，3气密NG，4注氦超时，5氦检异常，6电池泄漏，7注氦NG，8氦嘴泄漏）
LD TR0
AND>F(333) D402 D994  ; #3-1腔体测试漏率（Pa.m3/s_Float）, 泄漏率设定值（Pa.m3/s_Float）
ANDNOT H5.10  ; 空跑程序
ANDNOT H5.02  ; 氦检仪屏蔽
MOV(021) &3 D408  ; #3-1腔体测试结果（1 OK，2腔体泄漏，3气密NG，4注氦超时，5氦检异常，6电池泄漏，7注氦NG，8氦嘴泄漏）

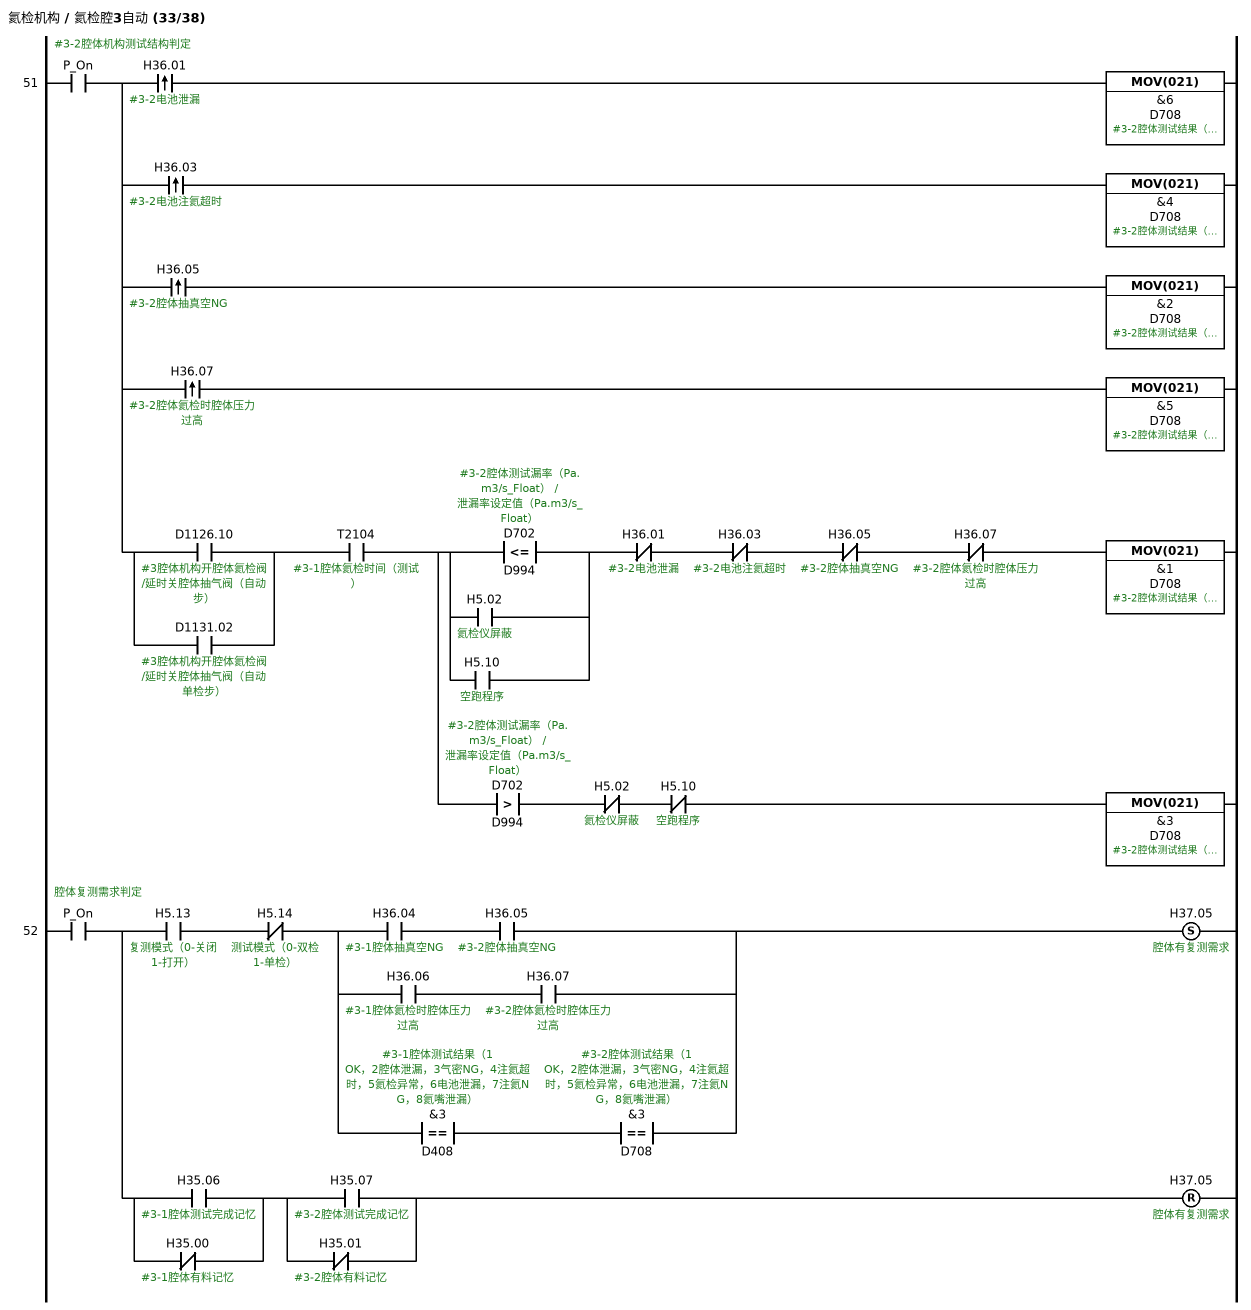
; rung 51: #3-2腔体机构测试结构判定
LD P_On
OUT TR0
@AND H36.01  ; #3-2电池泄漏
MOV(021) &6 D708  ; #3-2腔体测试结果（1 OK，2腔体泄漏，3气密NG，4注氦超时，5氦检异常，6电池泄漏，7注氦NG，8氦嘴泄漏）
LD TR0
@AND H36.03  ; #3-2电池注氦超时
MOV(021) &4 D708  ; #3-2腔体测试结果（1 OK，2腔体泄漏，3气密NG，4注氦超时，5氦检异常，6电池泄漏，7注氦NG，8氦嘴泄漏）
LD TR0
@AND H36.05  ; #3-2腔体抽真空NG
MOV(021) &2 D708  ; #3-2腔体测试结果（1 OK，2腔体泄漏，3气密NG，4注氦超时，5氦检异常，6电池泄漏，7注氦NG，8氦嘴泄漏）
LD TR0
@AND H36.07  ; #3-2腔体氦检时腔体压力过高
MOV(021) &5 D708  ; #3-2腔体测试结果（1 OK，2腔体泄漏，3气密NG，4注氦超时，5氦检异常，6电池泄漏，7注氦NG，8氦嘴泄漏）
LD TR0
LD D1126.10  ; #3腔体机构开腔体氦检阀/延时关腔体抽气阀（自动步）
OR D1131.02  ; #3腔体机构开腔体氦检阀/延时关腔体抽气阀（自动单检步）
ANDLD
AND T2104  ; #3-1腔体氦检时间（测试）
OUT TR0
LD<=F(332) D702 D994  ; #3-2腔体测试漏率（Pa.m3/s_Float）, 泄漏率设定值（Pa.m3/s_Float）
OR H5.02  ; 氦检仪屏蔽
OR H5.10  ; 空跑程序
ANDLD
ANDNOT H36.01  ; #3-2电池泄漏
ANDNOT H36.03  ; #3-2电池注氦超时
ANDNOT H36.05  ; #3-2腔体抽真空NG
ANDNOT H36.07  ; #3-2腔体氦检时腔体压力过高
MOV(021) &1 D708  ; #3-2腔体测试结果（1 OK，2腔体泄漏，3气密NG，4注氦超时，5氦检异常，6电池泄漏，7注氦NG，8氦嘴泄漏）
LD TR0
AND>F(333) D702 D994  ; #3-2腔体测试漏率（Pa.m3/s_Float）, 泄漏率设定值（Pa.m3/s_Float）
ANDNOT H5.02  ; 氦检仪屏蔽
ANDNOT H5.10  ; 空跑程序
MOV(021) &3 D708  ; #3-2腔体测试结果（1 OK，2腔体泄漏，3气密NG，4注氦超时，5氦检异常，6电池泄漏，7注氦NG，8氦嘴泄漏）
; rung 52: 腔体复测需求判定
LD P_On
OUT TR0
AND H5.13  ; 复测模式（0-关闭 1-打开）
ANDNOT H5.14  ; 测试模式（0-双检 1-单检）
LD H36.04  ; #3-1腔体抽真空NG
AND H36.05  ; #3-2腔体抽真空NG
LD H36.06  ; #3-1腔体氦检时腔体压力过高
AND H36.07  ; #3-2腔体氦检时腔体压力过高
ORLD
LD=(300) &3 D408  ; #3-1腔体测试结果（1 OK，2腔体泄漏，3气密NG，4注氦超时，5氦检异常，6电池泄漏，7注氦NG，8氦嘴泄漏）
AND=(300) &3 D708  ; #3-2腔体测试结果（1 OK，2腔体泄漏，3气密NG，4注氦超时，5氦检异常，6电池泄漏，7注氦NG，8氦嘴泄漏）
ORLD
ANDLD
SET H37.05  ; 腔体有复测需求
LD TR0
LD H35.06  ; #3-1腔体测试完成记忆
ORNOT H35.00  ; #3-1腔体有料记忆
ANDLD
LD H35.07  ; #3-2腔体测试完成记忆
ORNOT H35.01  ; #3-2腔体有料记忆
ANDLD
RSET H37.05  ; 腔体有复测需求

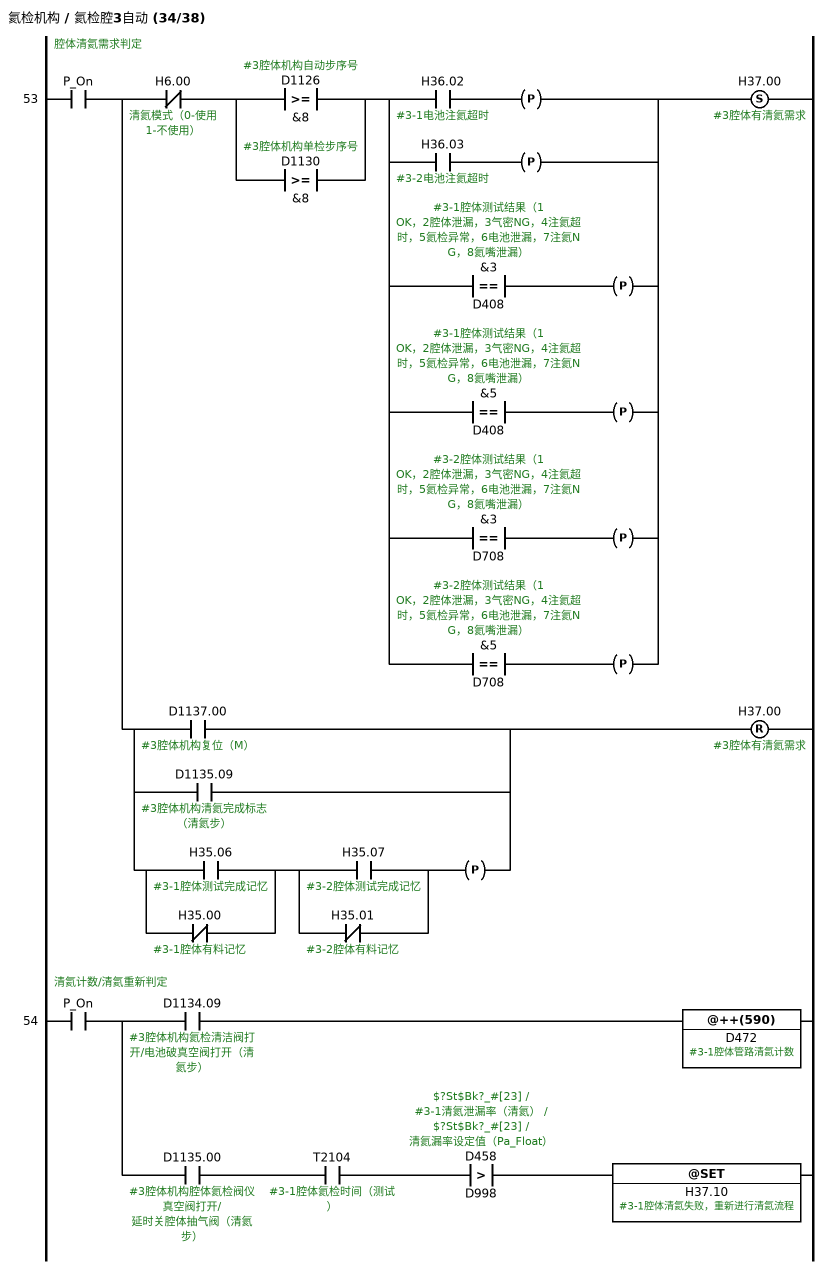
; rung 53: 腔体清氦需求判定
LD P_On
OUT TR0
ANDNOT H6.00  ; 清氦模式（0-使用 1-不使用）
LD>=L(326) D1126 &8  ; #3腔体机构自动步序号
OR>=L(326) D1130 &8  ; #3腔体机构单检步序号
ANDLD
LD H36.02  ; #3-1电池注氦超时
UP(521)
LD H36.03  ; #3-2电池注氦超时
UP(521)
ORLD
LD=(300) &3 D408  ; #3-1腔体测试结果（1 OK，2腔体泄漏，3气密NG，4注氦超时，5氦检异常，6电池泄漏，7注氦NG，8氦嘴泄漏）
UP(521)
ORLD
LD=(300) &5 D408  ; #3-1腔体测试结果（1 OK，2腔体泄漏，3气密NG，4注氦超时，5氦检异常，6电池泄漏，7注氦NG，8氦嘴泄漏）
UP(521)
ORLD
LD=(300) &3 D708  ; #3-2腔体测试结果（1 OK，2腔体泄漏，3气密NG，4注氦超时，5氦检异常，6电池泄漏，7注氦NG，8氦嘴泄漏）
UP(521)
ORLD
LD=(300) &5 D708  ; #3-2腔体测试结果（1 OK，2腔体泄漏，3气密NG，4注氦超时，5氦检异常，6电池泄漏，7注氦NG，8氦嘴泄漏）
UP(521)
ORLD
ANDLD
SET H37.00  ; #3腔体有清氦需求
LD TR0
LD D1137.00  ; #3腔体机构复位（M）
OR D1135.09  ; #3腔体机构清氦完成标志（清氦步）
LD H35.06  ; #3-1腔体测试完成记忆
ORNOT H35.00  ; #3-1腔体有料记忆
LD H35.07  ; #3-2腔体测试完成记忆
ORNOT H35.01  ; #3-2腔体有料记忆
ANDLD
UP(521)
ORLD
ANDLD
RSET H37.00  ; #3腔体有清氦需求
; rung 54: 清氦计数/清氦重新判定
LD P_On
OUT TR0
AND D1134.09  ; #3腔体机构氦检清洁阀打开/电池破真空阀打开（清氦步）
@++(590) D472  ; #3-1腔体管路清氦计数
LD TR0
AND D1135.00  ; #3腔体机构腔体氦检阀仪真空阀打开/延时关腔体抽气阀（清氦步）
AND T2104  ; #3-1腔体氦检时间（测试）
AND>F(333) D458 D998  ; $?St$Bk?_#[23] / #3-1清氦泄漏率（清氦） / $?St$Bk?_#[23], 清氦漏率设定值（Pa_Float）
@SET H37.10  ; #3-1腔体清氦失败，重新进行清氦流程

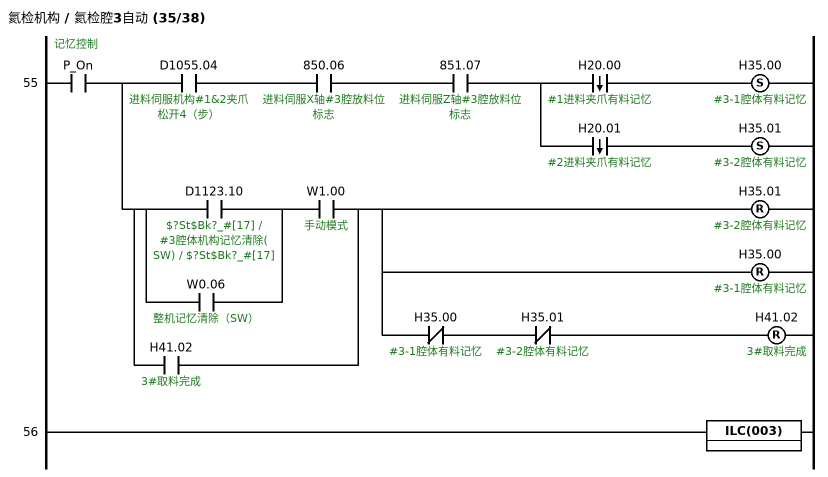
; rung 55: 记忆控制
LD P_On
OUT TR0
AND D1055.04  ; 进料伺服机构#1&2夹爪松开4（步）
AND 850.06  ; 进料伺服X轴#3腔放料位标志
AND 851.07  ; 进料伺服Z轴#3腔放料位标志
OUT TR1
%AND H20.00  ; #1进料夹爪有料记忆
SET H35.00  ; #3-1腔体有料记忆
LD TR1
%AND H20.01  ; #2进料夹爪有料记忆
SET H35.01  ; #3-2腔体有料记忆
LD TR0
LD D1123.10  ; $?St$Bk?_#[17] / #3腔体机构记忆清除(SW) / $?St$Bk?_#[17]
OR W0.06  ; 整机记忆清除（SW）
AND W1.00  ; 手动模式
OR H41.02  ; 3#取料完成
ANDLD
RSET H35.01  ; #3-2腔体有料记忆
RSET H35.00  ; #3-1腔体有料记忆
ANDNOT H35.00  ; #3-1腔体有料记忆
ANDNOT H35.01  ; #3-2腔体有料记忆
RSET H41.02  ; 3#取料完成
; rung 56
ILC(003)

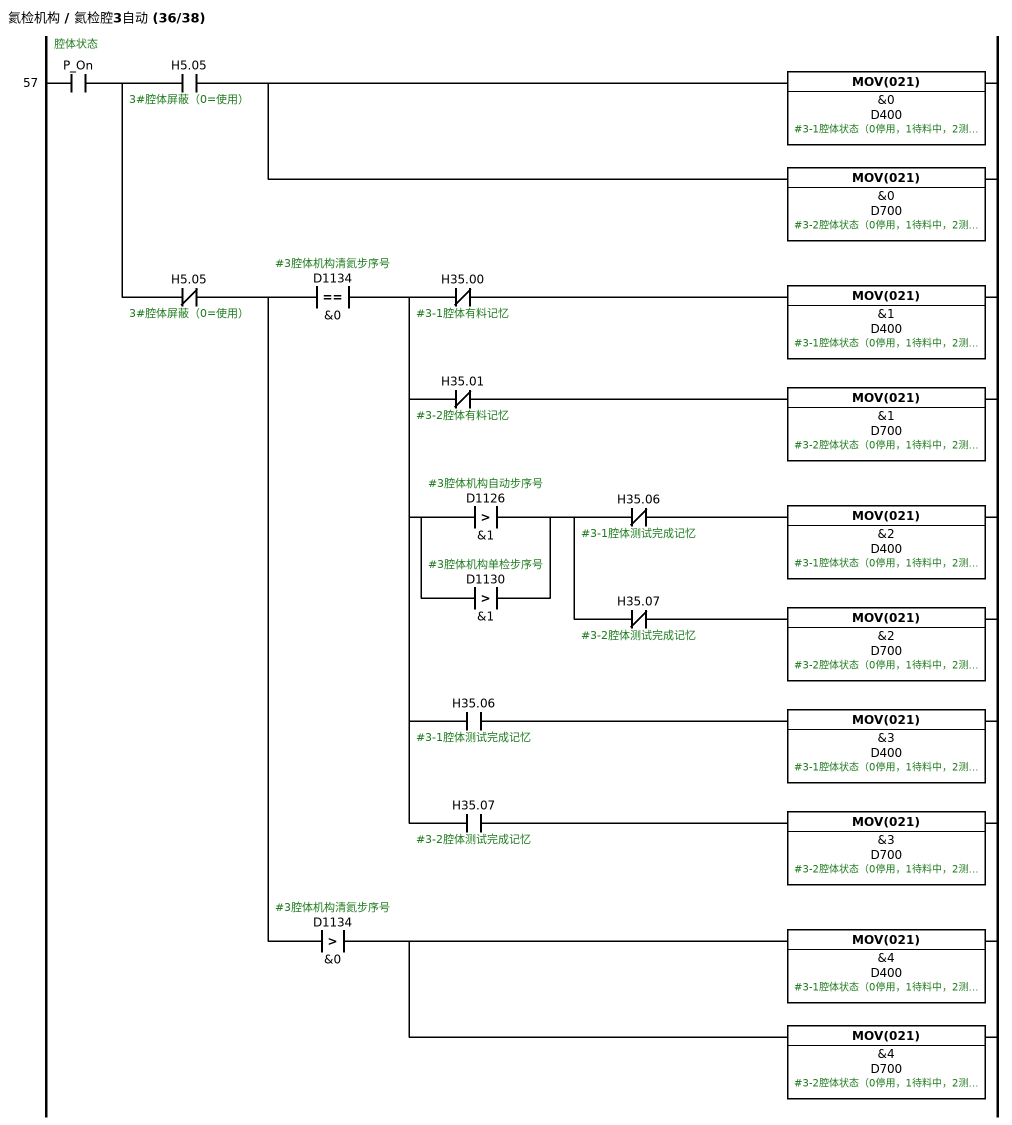
; rung 57: 腔体状态
LD P_On
OUT TR0
AND H5.05  ; 3#腔体屏蔽（0=使用）
MOV(021) &0 D400  ; #3-1腔体状态（0停用，1待料中，2测试中，3测试完成，4-清氦中）
MOV(021) &0 D700  ; #3-2腔体状态（0停用，1待料中，2测试中，3测试完成，4-清氦中）
LD TR0
ANDNOT H5.05  ; 3#腔体屏蔽（0=使用）
OUT TR0
AND=L(301) D1134 &0  ; #3腔体机构清氦步序号
OUT TR1
ANDNOT H35.00  ; #3-1腔体有料记忆
MOV(021) &1 D400  ; #3-1腔体状态（0停用，1待料中，2测试中，3测试完成，4-清氦中）
LD TR1
ANDNOT H35.01  ; #3-2腔体有料记忆
MOV(021) &1 D700  ; #3-2腔体状态（0停用，1待料中，2测试中，3测试完成，4-清氦中）
LD TR1
LD>L(321) D1126 &1  ; #3腔体机构自动步序号
OR>L(321) D1130 &1  ; #3腔体机构单检步序号
ANDLD
OUT TR2
ANDNOT H35.06  ; #3-1腔体测试完成记忆
MOV(021) &2 D400  ; #3-1腔体状态（0停用，1待料中，2测试中，3测试完成，4-清氦中）
LD TR2
ANDNOT H35.07  ; #3-2腔体测试完成记忆
MOV(021) &2 D700  ; #3-2腔体状态（0停用，1待料中，2测试中，3测试完成，4-清氦中）
LD TR1
AND H35.06  ; #3-1腔体测试完成记忆
MOV(021) &3 D400  ; #3-1腔体状态（0停用，1待料中，2测试中，3测试完成，4-清氦中）
LD TR1
AND H35.07  ; #3-2腔体测试完成记忆
MOV(021) &3 D700  ; #3-2腔体状态（0停用，1待料中，2测试中，3测试完成，4-清氦中）
LD TR0
AND>L(321) D1134 &0  ; #3腔体机构清氦步序号
MOV(021) &4 D400  ; #3-1腔体状态（0停用，1待料中，2测试中，3测试完成，4-清氦中）
MOV(021) &4 D700  ; #3-2腔体状态（0停用，1待料中，2测试中，3测试完成，4-清氦中）

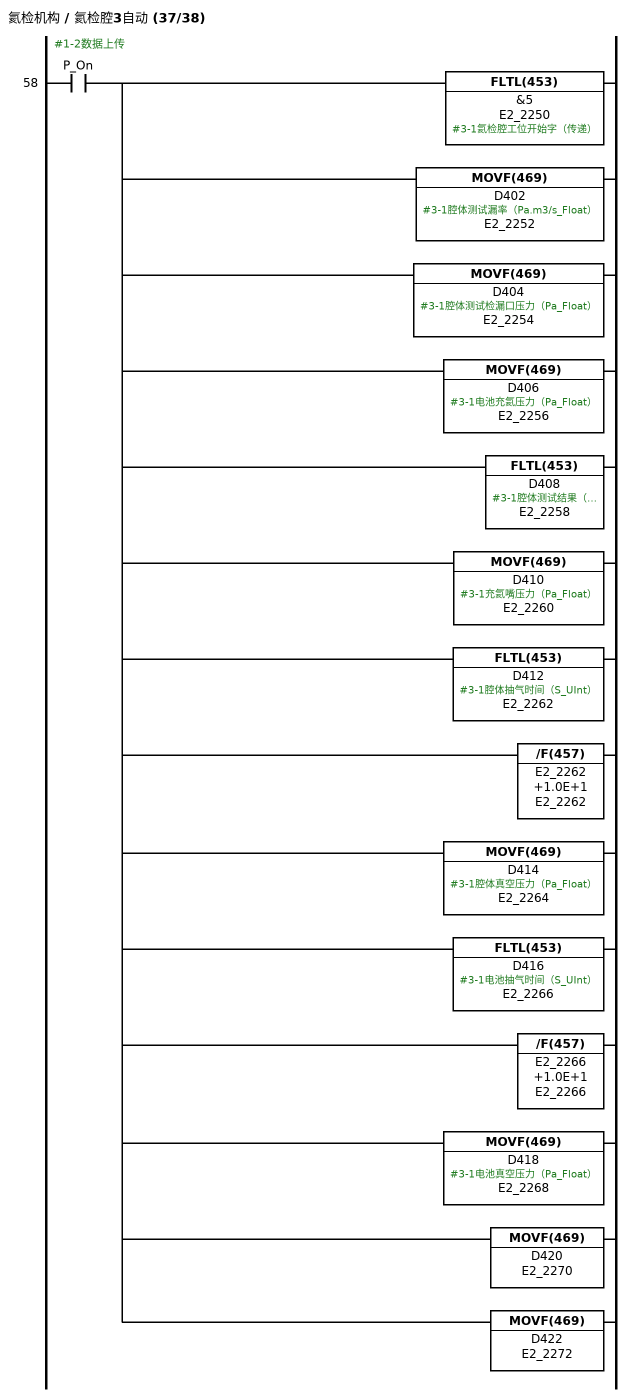
; rung 58: #1-2数据上传
LD P_On
FLTL(453) &5 E2_2250  ; #3-1氦检腔工位开始字（传递）
MOVF(469) D402 E2_2252  ; #3-1腔体测试漏率（Pa.m3/s_Float）
MOVF(469) D404 E2_2254  ; #3-1腔体测试检漏口压力（Pa_Float）
MOVF(469) D406 E2_2256  ; #3-1电池充氦压力（Pa_Float）
FLTL(453) D408 E2_2258  ; #3-1腔体测试结果（1 OK，2腔体泄漏，3气密NG，4注氦超时，5氦检异常，6电池泄漏，7注氦NG，8氦嘴泄漏）
MOVF(469) D410 E2_2260  ; #3-1充氦嘴压力（Pa_Float）
FLTL(453) D412 E2_2262  ; #3-1腔体抽气时间（S_UInt）
/F(457) E2_2262 +1.0E+1 E2_2262
MOVF(469) D414 E2_2264  ; #3-1腔体真空压力（Pa_Float）
FLTL(453) D416 E2_2266  ; #3-1电池抽气时间（S_UInt）
/F(457) E2_2266 +1.0E+1 E2_2266
MOVF(469) D418 E2_2268  ; #3-1电池真空压力（Pa_Float）
MOVF(469) D420 E2_2270
MOVF(469) D422 E2_2272

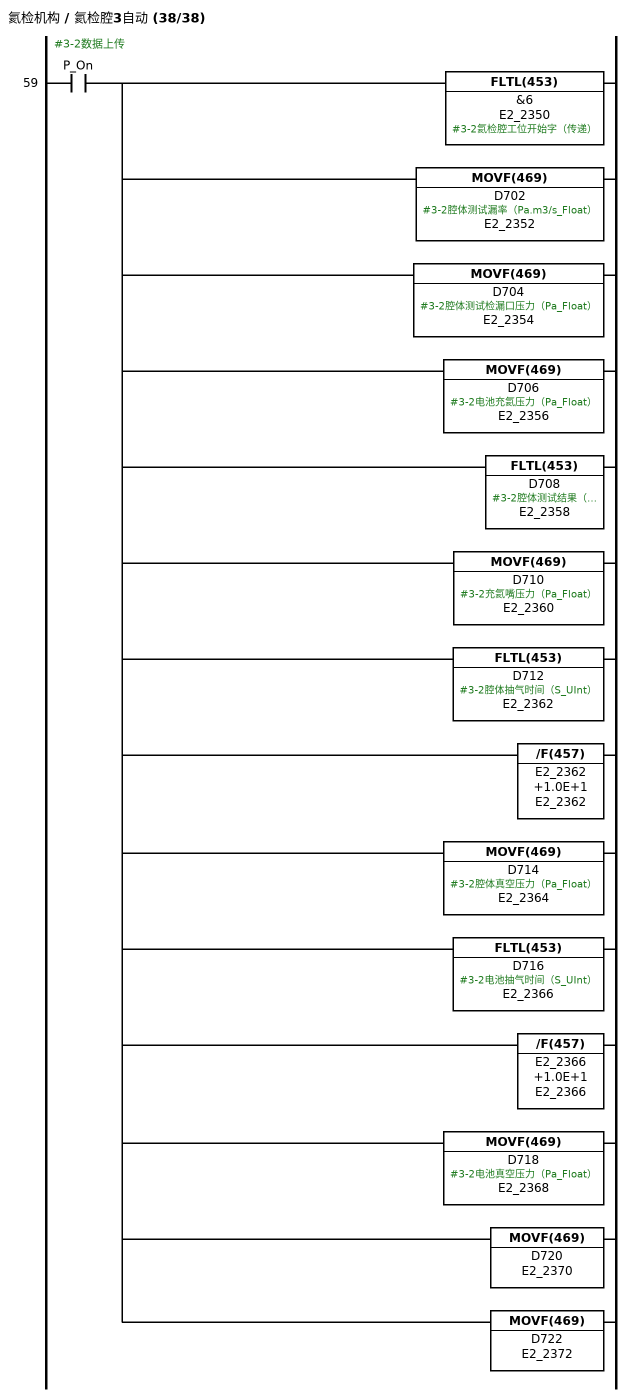
; rung 59: #3-2数据上传
LD P_On
FLTL(453) &6 E2_2350  ; #3-2氦检腔工位开始字（传递）
MOVF(469) D702 E2_2352  ; #3-2腔体测试漏率（Pa.m3/s_Float）
MOVF(469) D704 E2_2354  ; #3-2腔体测试检漏口压力（Pa_Float）
MOVF(469) D706 E2_2356  ; #3-2电池充氦压力（Pa_Float）
FLTL(453) D708 E2_2358  ; #3-2腔体测试结果（1 OK，2腔体泄漏，3气密NG，4注氦超时，5氦检异常，6电池泄漏，7注氦NG，8氦嘴泄漏）
MOVF(469) D710 E2_2360  ; #3-2充氦嘴压力（Pa_Float）
FLTL(453) D712 E2_2362  ; #3-2腔体抽气时间（S_UInt）
/F(457) E2_2362 +1.0E+1 E2_2362
MOVF(469) D714 E2_2364  ; #3-2腔体真空压力（Pa_Float）
FLTL(453) D716 E2_2366  ; #3-2电池抽气时间（S_UInt）
/F(457) E2_2366 +1.0E+1 E2_2366
MOVF(469) D718 E2_2368  ; #3-2电池真空压力（Pa_Float）
MOVF(469) D720 E2_2370
MOVF(469) D722 E2_2372

### Section 工站复位

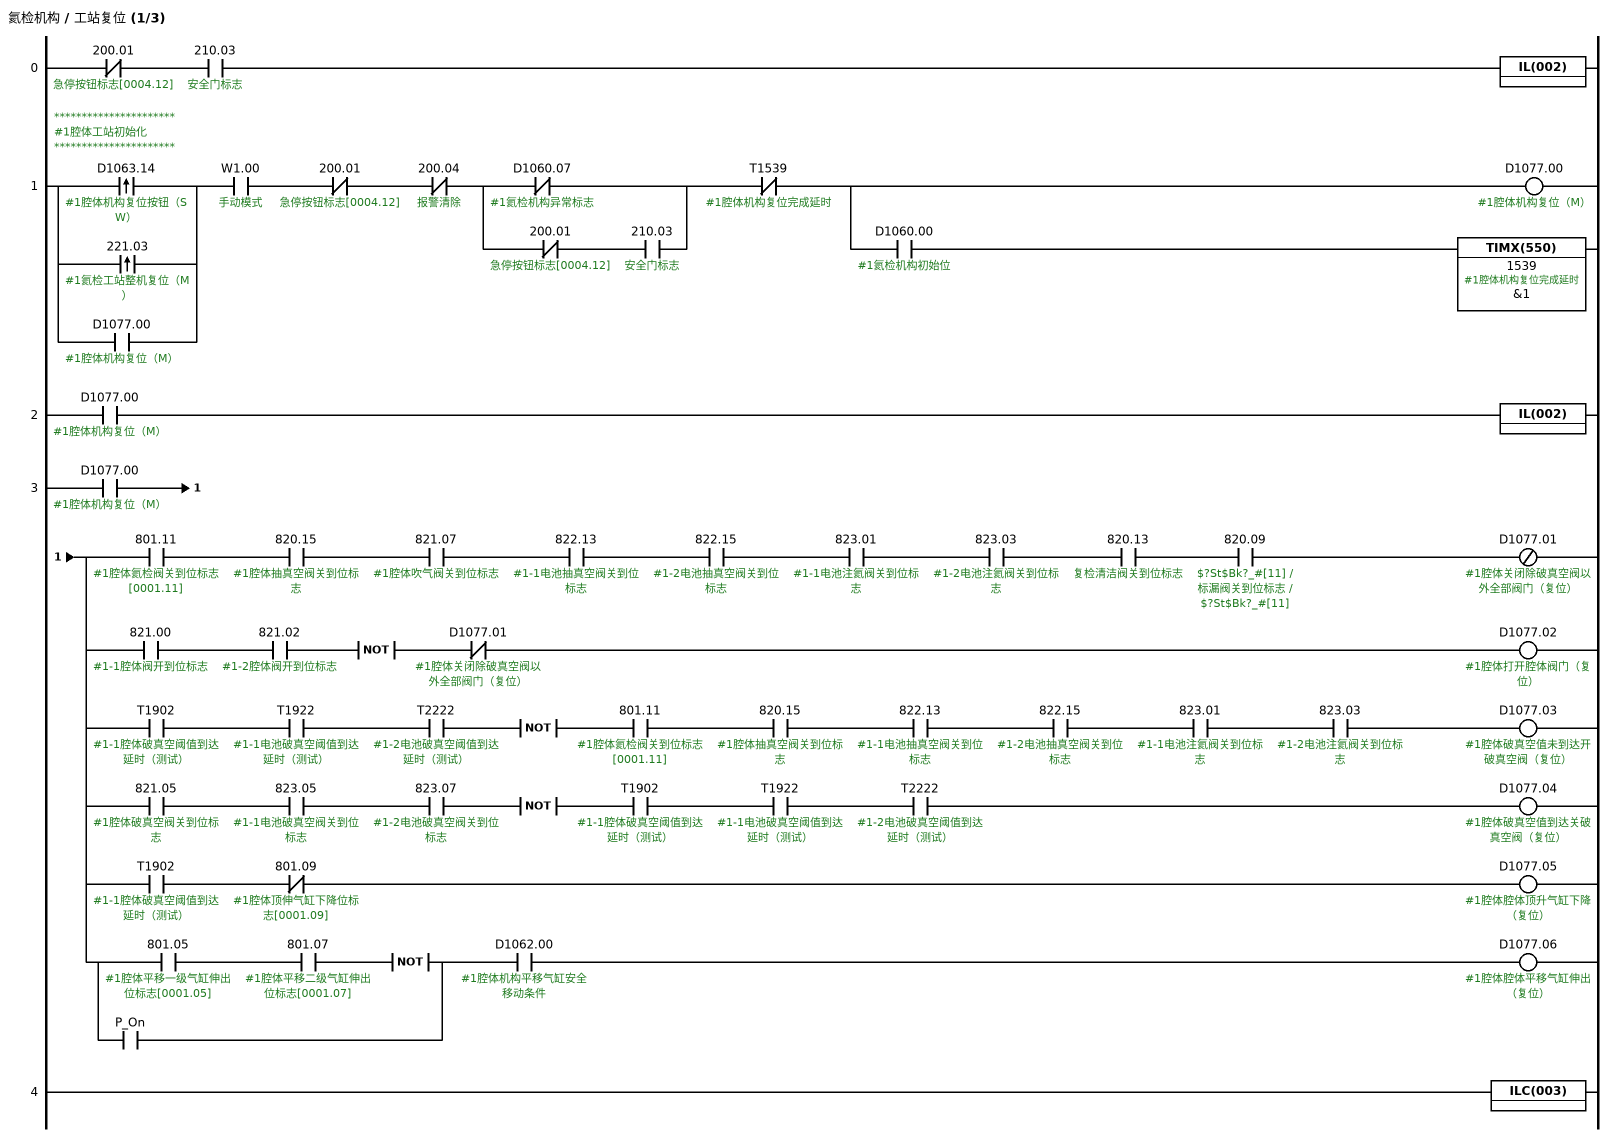
; rung 0
LDNOT 200.01  ; 急停按钮标志[0004.12]
AND 210.03  ; 安全门标志
IL(002)
; rung 1: ********************** / #1腔体工站初始化 / **********************
@LD D1063.14  ; #1腔体机构复位按钮（SW）
@OR 221.03  ; #1氦检工站整机复位（M）
OR D1077.00  ; #1腔体机构复位（M）
AND W1.00  ; 手动模式
ANDNOT 200.01  ; 急停按钮标志[0004.12]
ANDNOT 200.04  ; 报警清除
LDNOT D1060.07  ; #1氦检机构异常标志
LDNOT 200.01  ; 急停按钮标志[0004.12]
AND 210.03  ; 安全门标志
ORLD
ANDLD
ANDNOT T1539  ; #1腔体机构复位完成延时
OUT D1077.00  ; #1腔体机构复位（M）
AND D1060.00  ; #1氦检机构初始位
TIMX(550) 1539 &1  ; #1腔体机构复位完成延时
; rung 2
LD D1077.00  ; #1腔体机构复位（M）
IL(002)
; rung 3
LD D1077.00  ; #1腔体机构复位（M）
OUT TR0
AND 801.11  ; #1腔体氦检阀关到位标志[0001.11]
AND 820.15  ; #1腔体抽真空阀关到位标志
AND 821.07  ; #1腔体吹气阀关到位标志
AND 822.13  ; #1-1电池抽真空阀关到位标志
AND 822.15  ; #1-2电池抽真空阀关到位标志
AND 823.01  ; #1-1电池注氦阀关到位标志
AND 823.03  ; #1-2电池注氦阀关到位标志
AND 820.13  ; 复检清洁阀关到位标志
AND 820.09  ; $?St$Bk?_#[11] / 标漏阀关到位标志 / $?St$Bk?_#[11]
OUTNOT D1077.01  ; #1腔体关闭除破真空阀以外全部阀门（复位）
LD TR0
AND 821.00  ; #1-1腔体阀开到位标志
AND 821.02  ; #1-2腔体阀开到位标志
NOT(520)
ANDNOT D1077.01  ; #1腔体关闭除破真空阀以外全部阀门（复位）
OUT D1077.02  ; #1腔体打开腔体阀门（复位）
LD TR0
AND T1902  ; #1-1腔体破真空阈值到达延时（测试）
AND T1922  ; #1-1电池破真空阈值到达延时（测试）
AND T2222  ; #1-2电池破真空阈值到达延时（测试）
NOT(520)
AND 801.11  ; #1腔体氦检阀关到位标志[0001.11]
AND 820.15  ; #1腔体抽真空阀关到位标志
AND 822.13  ; #1-1电池抽真空阀关到位标志
AND 822.15  ; #1-2电池抽真空阀关到位标志
AND 823.01  ; #1-1电池注氦阀关到位标志
AND 823.03  ; #1-2电池注氦阀关到位标志
OUT D1077.03  ; #1腔体破真空值未到达开破真空阀（复位）
LD TR0
AND 821.05  ; #1腔体破真空阀关到位标志
AND 823.05  ; #1-1电池破真空阀关到位标志
AND 823.07  ; #1-2电池破真空阀关到位标志
NOT(520)
AND T1902  ; #1-1腔体破真空阈值到达延时（测试）
AND T1922  ; #1-1电池破真空阈值到达延时（测试）
AND T2222  ; #1-2电池破真空阈值到达延时（测试）
OUT D1077.04  ; #1腔体破真空值到达关破真空阀（复位）
LD TR0
AND T1902  ; #1-1腔体破真空阈值到达延时（测试）
ANDNOT 801.09  ; #1腔体顶伸气缸下降位标志[0001.09]
OUT D1077.05  ; #1腔体腔体顶升气缸下降（复位）
LD TR0
LD 801.05  ; #1腔体平移一级气缸伸出位标志[0001.05]
AND 801.07  ; #1腔体平移二级气缸伸出位标志[0001.07]
NOT(520)
OR P_On
ANDLD
AND D1062.00  ; #1腔体机构平移气缸安全移动条件
OUT D1077.06  ; #1腔体腔体平移气缸伸出（复位）
; rung 4
ILC(003)

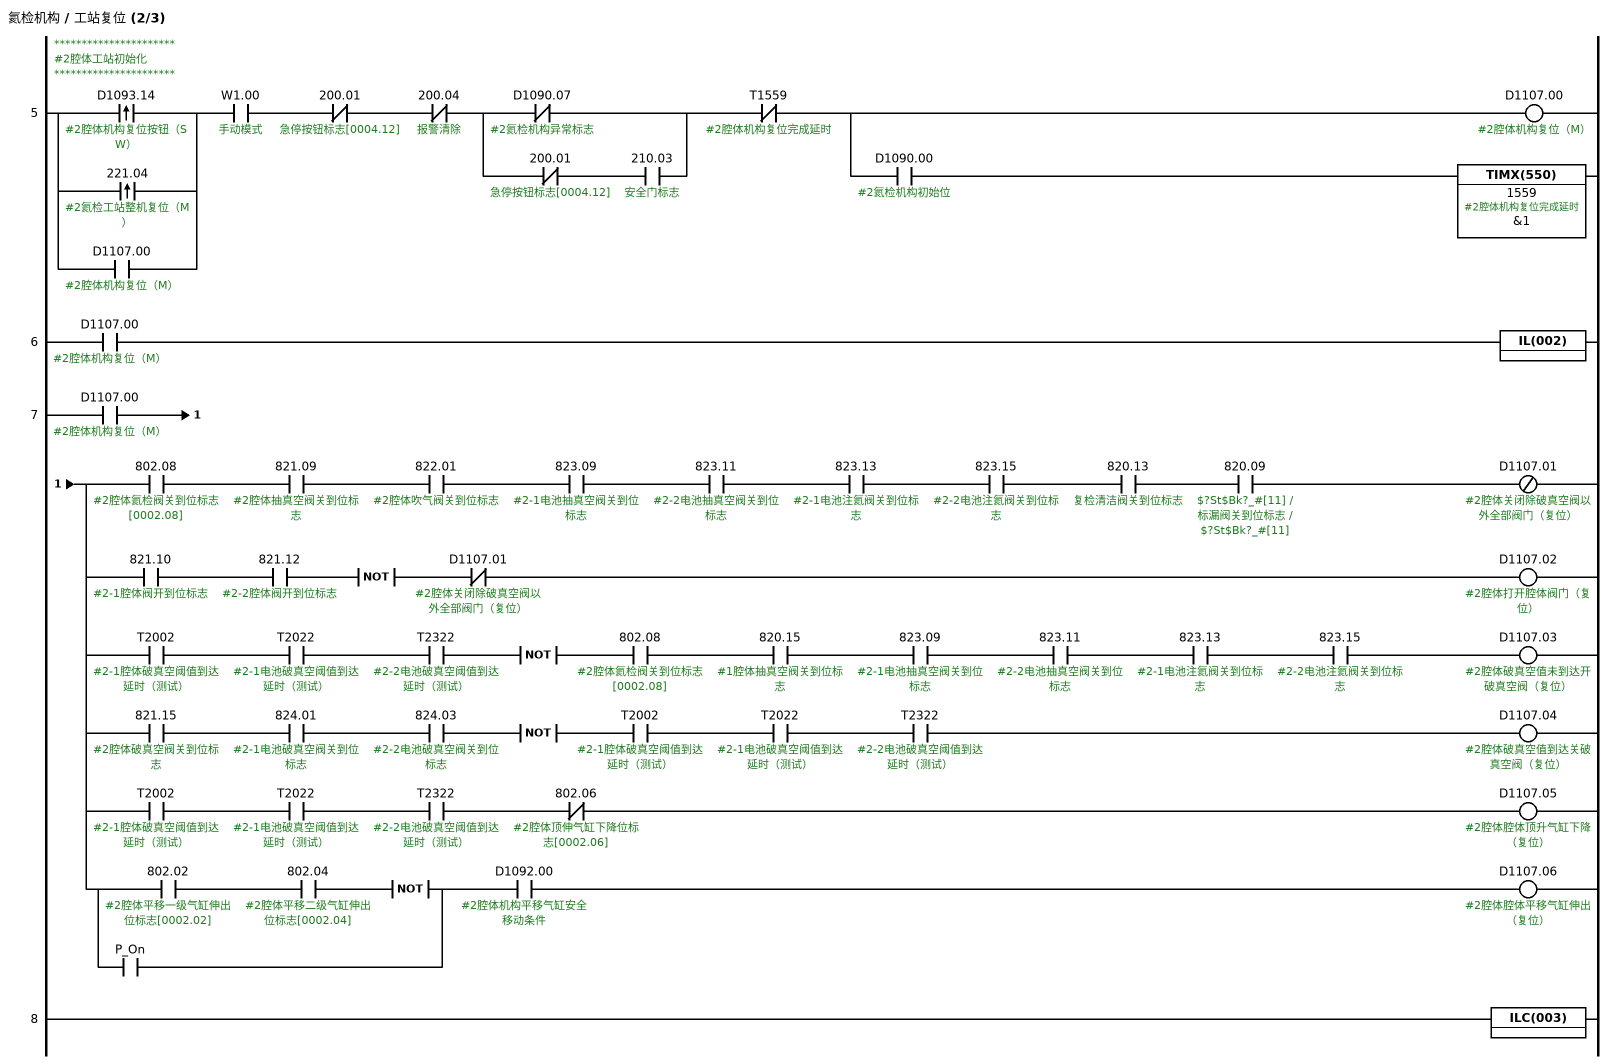
; rung 5: ********************** / #2腔体工站初始化 / **********************
@LD D1093.14  ; #2腔体机构复位按钮（SW）
@OR 221.04  ; #2氦检工站整机复位（M）
OR D1107.00  ; #2腔体机构复位（M）
AND W1.00  ; 手动模式
ANDNOT 200.01  ; 急停按钮标志[0004.12]
ANDNOT 200.04  ; 报警清除
LDNOT D1090.07  ; #2氦检机构异常标志
LDNOT 200.01  ; 急停按钮标志[0004.12]
AND 210.03  ; 安全门标志
ORLD
ANDLD
ANDNOT T1559  ; #2腔体机构复位完成延时
OUT D1107.00  ; #2腔体机构复位（M）
AND D1090.00  ; #2氦检机构初始位
TIMX(550) 1559 &1  ; #2腔体机构复位完成延时
; rung 6
LD D1107.00  ; #2腔体机构复位（M）
IL(002)
; rung 7
LD D1107.00  ; #2腔体机构复位（M）
OUT TR0
AND 802.08  ; #2腔体氦检阀关到位标志[0002.08]
AND 821.09  ; #2腔体抽真空阀关到位标志
AND 822.01  ; #2腔体吹气阀关到位标志
AND 823.09  ; #2-1电池抽真空阀关到位标志
AND 823.11  ; #2-2电池抽真空阀关到位标志
AND 823.13  ; #2-1电池注氦阀关到位标志
AND 823.15  ; #2-2电池注氦阀关到位标志
AND 820.13  ; 复检清洁阀关到位标志
AND 820.09  ; $?St$Bk?_#[11] / 标漏阀关到位标志 / $?St$Bk?_#[11]
OUTNOT D1107.01  ; #2腔体关闭除破真空阀以外全部阀门（复位）
LD TR0
AND 821.10  ; #2-1腔体阀开到位标志
AND 821.12  ; #2-2腔体阀开到位标志
NOT(520)
ANDNOT D1107.01  ; #2腔体关闭除破真空阀以外全部阀门（复位）
OUT D1107.02  ; #2腔体打开腔体阀门（复位）
LD TR0
AND T2002  ; #2-1腔体破真空阈值到达延时（测试）
AND T2022  ; #2-1电池破真空阈值到达延时（测试）
AND T2322  ; #2-2电池破真空阈值到达延时（测试）
NOT(520)
AND 802.08  ; #2腔体氦检阀关到位标志[0002.08]
AND 820.15  ; #1腔体抽真空阀关到位标志
AND 823.09  ; #2-1电池抽真空阀关到位标志
AND 823.11  ; #2-2电池抽真空阀关到位标志
AND 823.13  ; #2-1电池注氦阀关到位标志
AND 823.15  ; #2-2电池注氦阀关到位标志
OUT D1107.03  ; #2腔体破真空值未到达开破真空阀（复位）
LD TR0
AND 821.15  ; #2腔体破真空阀关到位标志
AND 824.01  ; #2-1电池破真空阀关到位标志
AND 824.03  ; #2-2电池破真空阀关到位标志
NOT(520)
AND T2002  ; #2-1腔体破真空阈值到达延时（测试）
AND T2022  ; #2-1电池破真空阈值到达延时（测试）
AND T2322  ; #2-2电池破真空阈值到达延时（测试）
OUT D1107.04  ; #2腔体破真空值到达关破真空阀（复位）
LD TR0
AND T2002  ; #2-1腔体破真空阈值到达延时（测试）
AND T2022  ; #2-1电池破真空阈值到达延时（测试）
AND T2322  ; #2-2电池破真空阈值到达延时（测试）
ANDNOT 802.06  ; #2腔体顶伸气缸下降位标志[0002.06]
OUT D1107.05  ; #2腔体腔体顶升气缸下降（复位）
LD TR0
LD 802.02  ; #2腔体平移一级气缸伸出位标志[0002.02]
AND 802.04  ; #2腔体平移二级气缸伸出位标志[0002.04]
NOT(520)
OR P_On
ANDLD
AND D1092.00  ; #2腔体机构平移气缸安全移动条件
OUT D1107.06  ; #2腔体腔体平移气缸伸出（复位）
; rung 8
ILC(003)

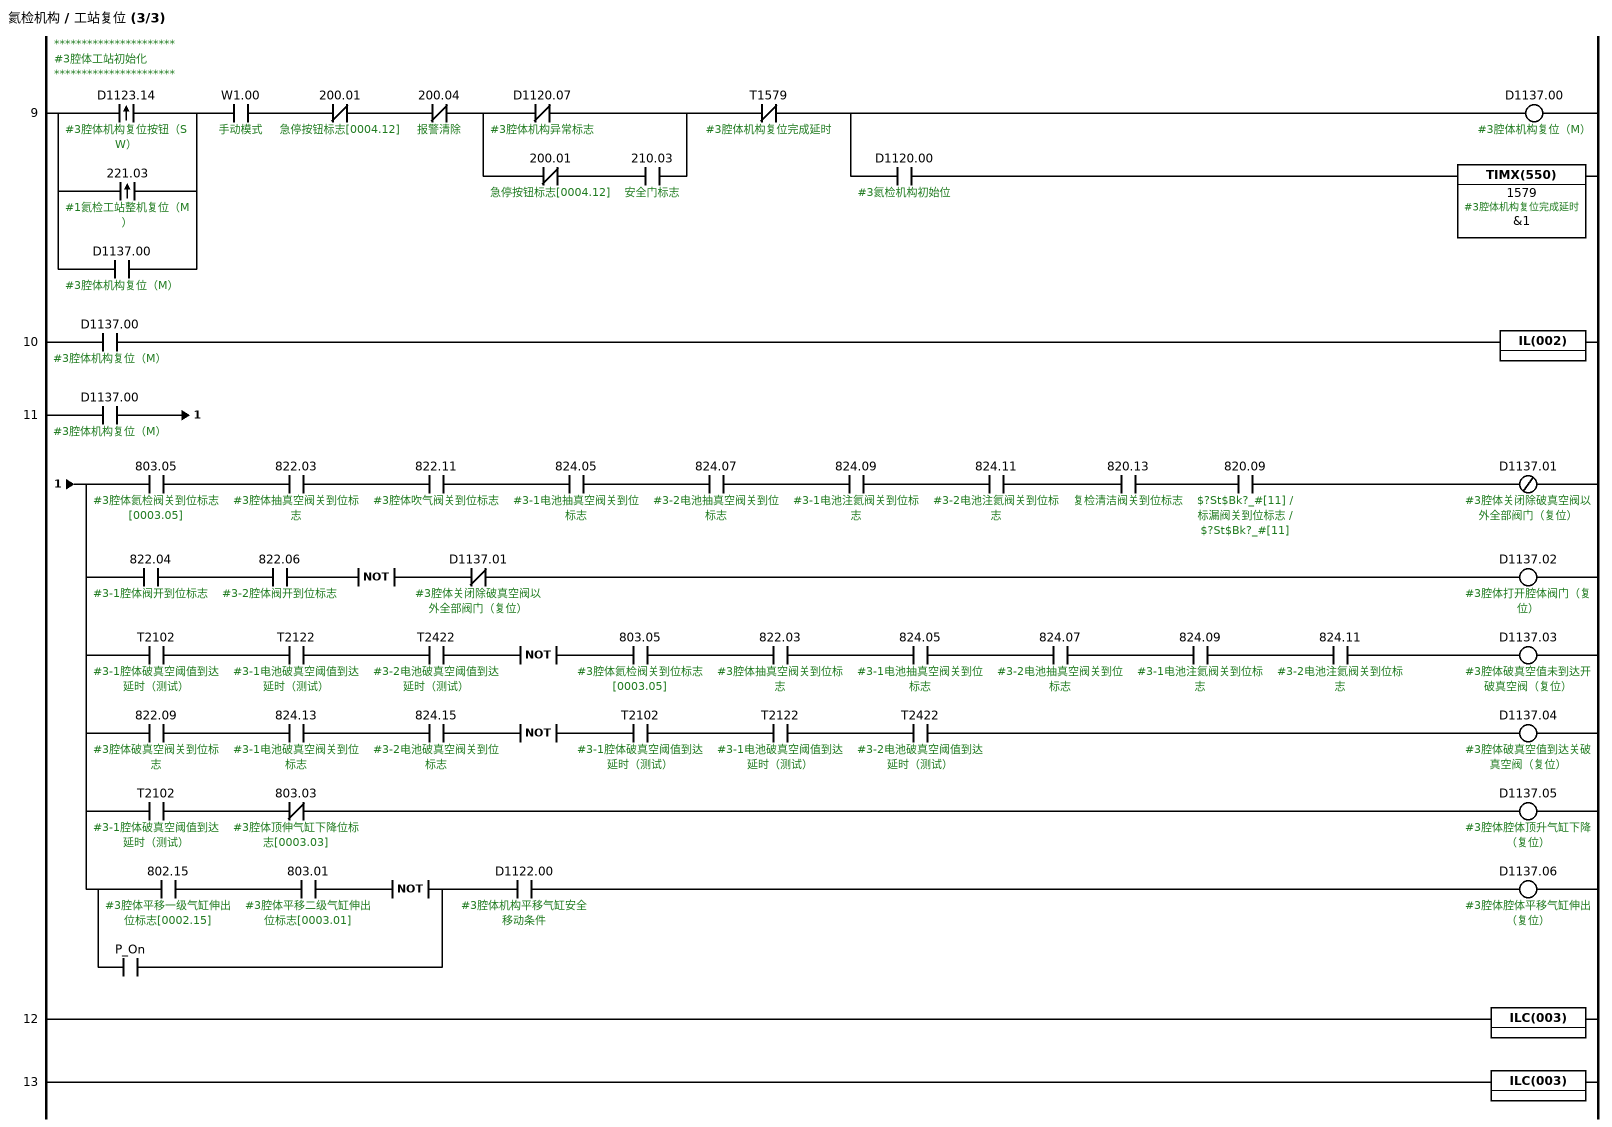
; rung 9: ********************** / #3腔体工站初始化 / **********************
@LD D1123.14  ; #3腔体机构复位按钮（SW）
@OR 221.03  ; #1氦检工站整机复位（M）
OR D1137.00  ; #3腔体机构复位（M）
AND W1.00  ; 手动模式
ANDNOT 200.01  ; 急停按钮标志[0004.12]
ANDNOT 200.04  ; 报警清除
LDNOT D1120.07  ; #3腔体机构异常标志
LDNOT 200.01  ; 急停按钮标志[0004.12]
AND 210.03  ; 安全门标志
ORLD
ANDLD
ANDNOT T1579  ; #3腔体机构复位完成延时
OUT D1137.00  ; #3腔体机构复位（M）
AND D1120.00  ; #3氦检机构初始位
TIMX(550) 1579 &1  ; #3腔体机构复位完成延时
; rung 10
LD D1137.00  ; #3腔体机构复位（M）
IL(002)
; rung 11
LD D1137.00  ; #3腔体机构复位（M）
OUT TR0
AND 803.05  ; #3腔体氦检阀关到位标志[0003.05]
AND 822.03  ; #3腔体抽真空阀关到位标志
AND 822.11  ; #3腔体吹气阀关到位标志
AND 824.05  ; #3-1电池抽真空阀关到位标志
AND 824.07  ; #3-2电池抽真空阀关到位标志
AND 824.09  ; #3-1电池注氦阀关到位标志
AND 824.11  ; #3-2电池注氦阀关到位标志
AND 820.13  ; 复检清洁阀关到位标志
AND 820.09  ; $?St$Bk?_#[11] / 标漏阀关到位标志 / $?St$Bk?_#[11]
OUTNOT D1137.01  ; #3腔体关闭除破真空阀以外全部阀门（复位）
LD TR0
AND 822.04  ; #3-1腔体阀开到位标志
AND 822.06  ; #3-2腔体阀开到位标志
NOT(520)
ANDNOT D1137.01  ; #3腔体关闭除破真空阀以外全部阀门（复位）
OUT D1137.02  ; #3腔体打开腔体阀门（复位）
LD TR0
AND T2102  ; #3-1腔体破真空阈值到达延时（测试）
AND T2122  ; #3-1电池破真空阈值到达延时（测试）
AND T2422  ; #3-2电池破真空阈值到达延时（测试）
NOT(520)
AND 803.05  ; #3腔体氦检阀关到位标志[0003.05]
AND 822.03  ; #3腔体抽真空阀关到位标志
AND 824.05  ; #3-1电池抽真空阀关到位标志
AND 824.07  ; #3-2电池抽真空阀关到位标志
AND 824.09  ; #3-1电池注氦阀关到位标志
AND 824.11  ; #3-2电池注氦阀关到位标志
OUT D1137.03  ; #3腔体破真空值未到达开破真空阀（复位）
LD TR0
AND 822.09  ; #3腔体破真空阀关到位标志
AND 824.13  ; #3-1电池破真空阀关到位标志
AND 824.15  ; #3-2电池破真空阀关到位标志
NOT(520)
AND T2102  ; #3-1腔体破真空阈值到达延时（测试）
AND T2122  ; #3-1电池破真空阈值到达延时（测试）
AND T2422  ; #3-2电池破真空阈值到达延时（测试）
OUT D1137.04  ; #3腔体破真空值到达关破真空阀（复位）
LD TR0
AND T2102  ; #3-1腔体破真空阈值到达延时（测试）
ANDNOT 803.03  ; #3腔体顶伸气缸下降位标志[0003.03]
OUT D1137.05  ; #3腔体腔体顶升气缸下降（复位）
LD TR0
LD 802.15  ; #3腔体平移一级气缸伸出位标志[0002.15]
AND 803.01  ; #3腔体平移二级气缸伸出位标志[0003.01]
NOT(520)
OR P_On
ANDLD
AND D1122.00  ; #3腔体机构平移气缸安全移动条件
OUT D1137.06  ; #3腔体腔体平移气缸伸出（复位）
; rung 12
ILC(003)
; rung 13
ILC(003)

### Section 腔体标漏

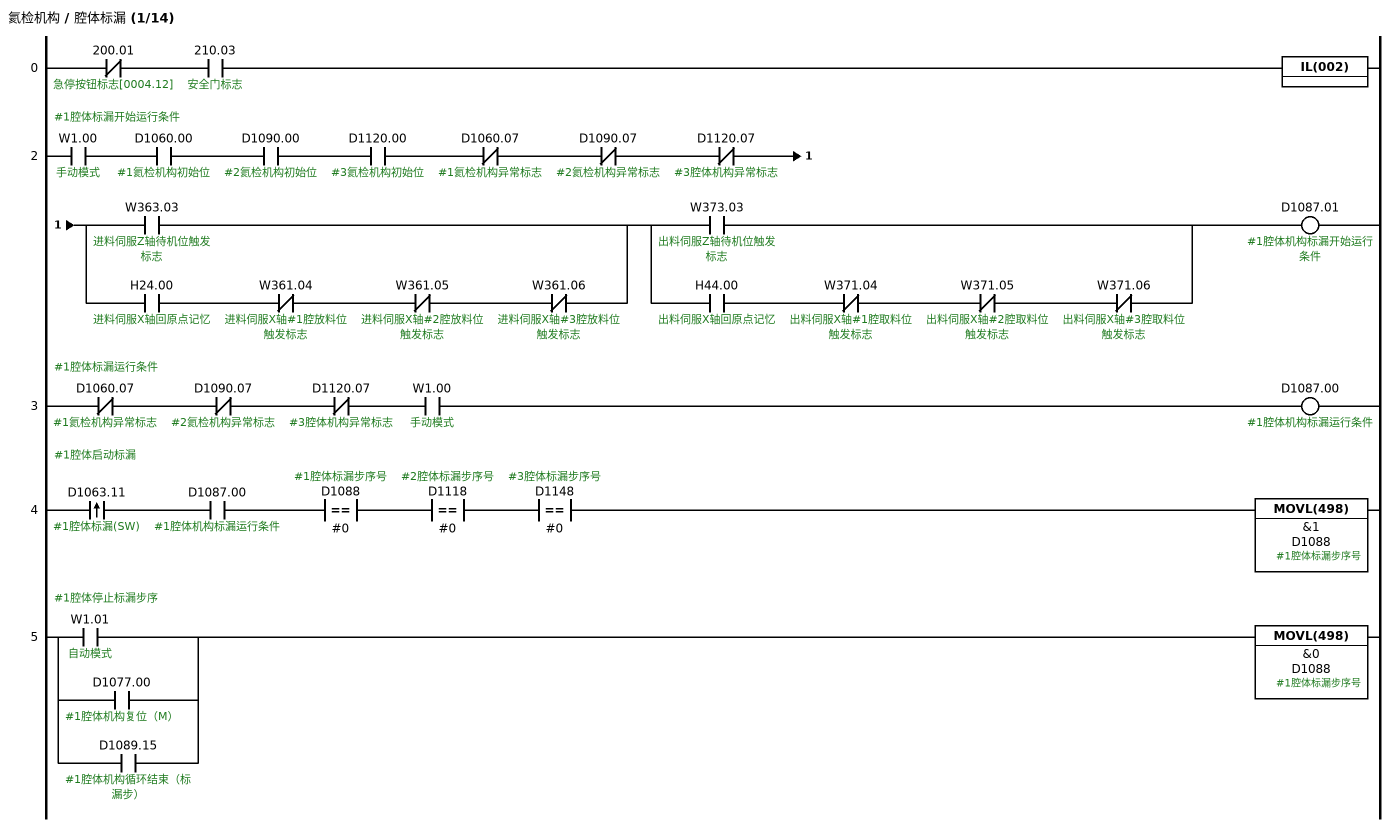
; rung 0
LDNOT 200.01  ; 急停按钮标志[0004.12]
AND 210.03  ; 安全门标志
IL(002)
; rung 1: ********************** / #1腔体标漏流程 / **********************
; rung 2: #1腔体标漏开始运行条件
LD W1.00  ; 手动模式
AND D1060.00  ; #1氦检机构初始位
AND D1090.00  ; #2氦检机构初始位
AND D1120.00  ; #3氦检机构初始位
ANDNOT D1060.07  ; #1氦检机构异常标志
ANDNOT D1090.07  ; #2氦检机构异常标志
ANDNOT D1120.07  ; #3腔体机构异常标志
LD W363.03  ; 进料伺服Z轴待机位触发标志
LD H24.00  ; 进料伺服X轴回原点记忆
ANDNOT W361.04  ; 进料伺服X轴#1腔放料位触发标志
ANDNOT W361.05  ; 进料伺服X轴#2腔放料位触发标志
ANDNOT W361.06  ; 进料伺服X轴#3腔放料位触发标志
ORLD
ANDLD
LD W373.03  ; 出料伺服Z轴待机位触发标志
LD H44.00  ; 出料伺服X轴回原点记忆
ANDNOT W371.04  ; 出料伺服X轴#1腔取料位触发标志
ANDNOT W371.05  ; 出料伺服X轴#2腔取料位触发标志
ANDNOT W371.06  ; 出料伺服X轴#3腔取料位触发标志
ORLD
ANDLD
OUT D1087.01  ; #1腔体机构标漏开始运行条件
; rung 3: #1腔体标漏运行条件
LDNOT D1060.07  ; #1氦检机构异常标志
ANDNOT D1090.07  ; #2氦检机构异常标志
ANDNOT D1120.07  ; #3腔体机构异常标志
AND W1.00  ; 手动模式
OUT D1087.00  ; #1腔体机构标漏运行条件
; rung 4: #1腔体启动标漏
@LD D1063.11  ; #1腔体标漏(SW)
AND D1087.00  ; #1腔体机构标漏运行条件
AND=L(301) D1088 #0  ; #1腔体标漏步序号
AND=L(301) D1118 #0  ; #2腔体标漏步序号
AND=L(301) D1148 #0  ; #3腔体标漏步序号
MOVL(498) &1 D1088  ; #1腔体标漏步序号
; rung 5: #1腔体停止标漏步序
LD W1.01  ; 自动模式
OR D1077.00  ; #1腔体机构复位（M）
OR D1089.15  ; #1腔体机构循环结束（标漏步）
MOVL(498) &0 D1088  ; #1腔体标漏步序号

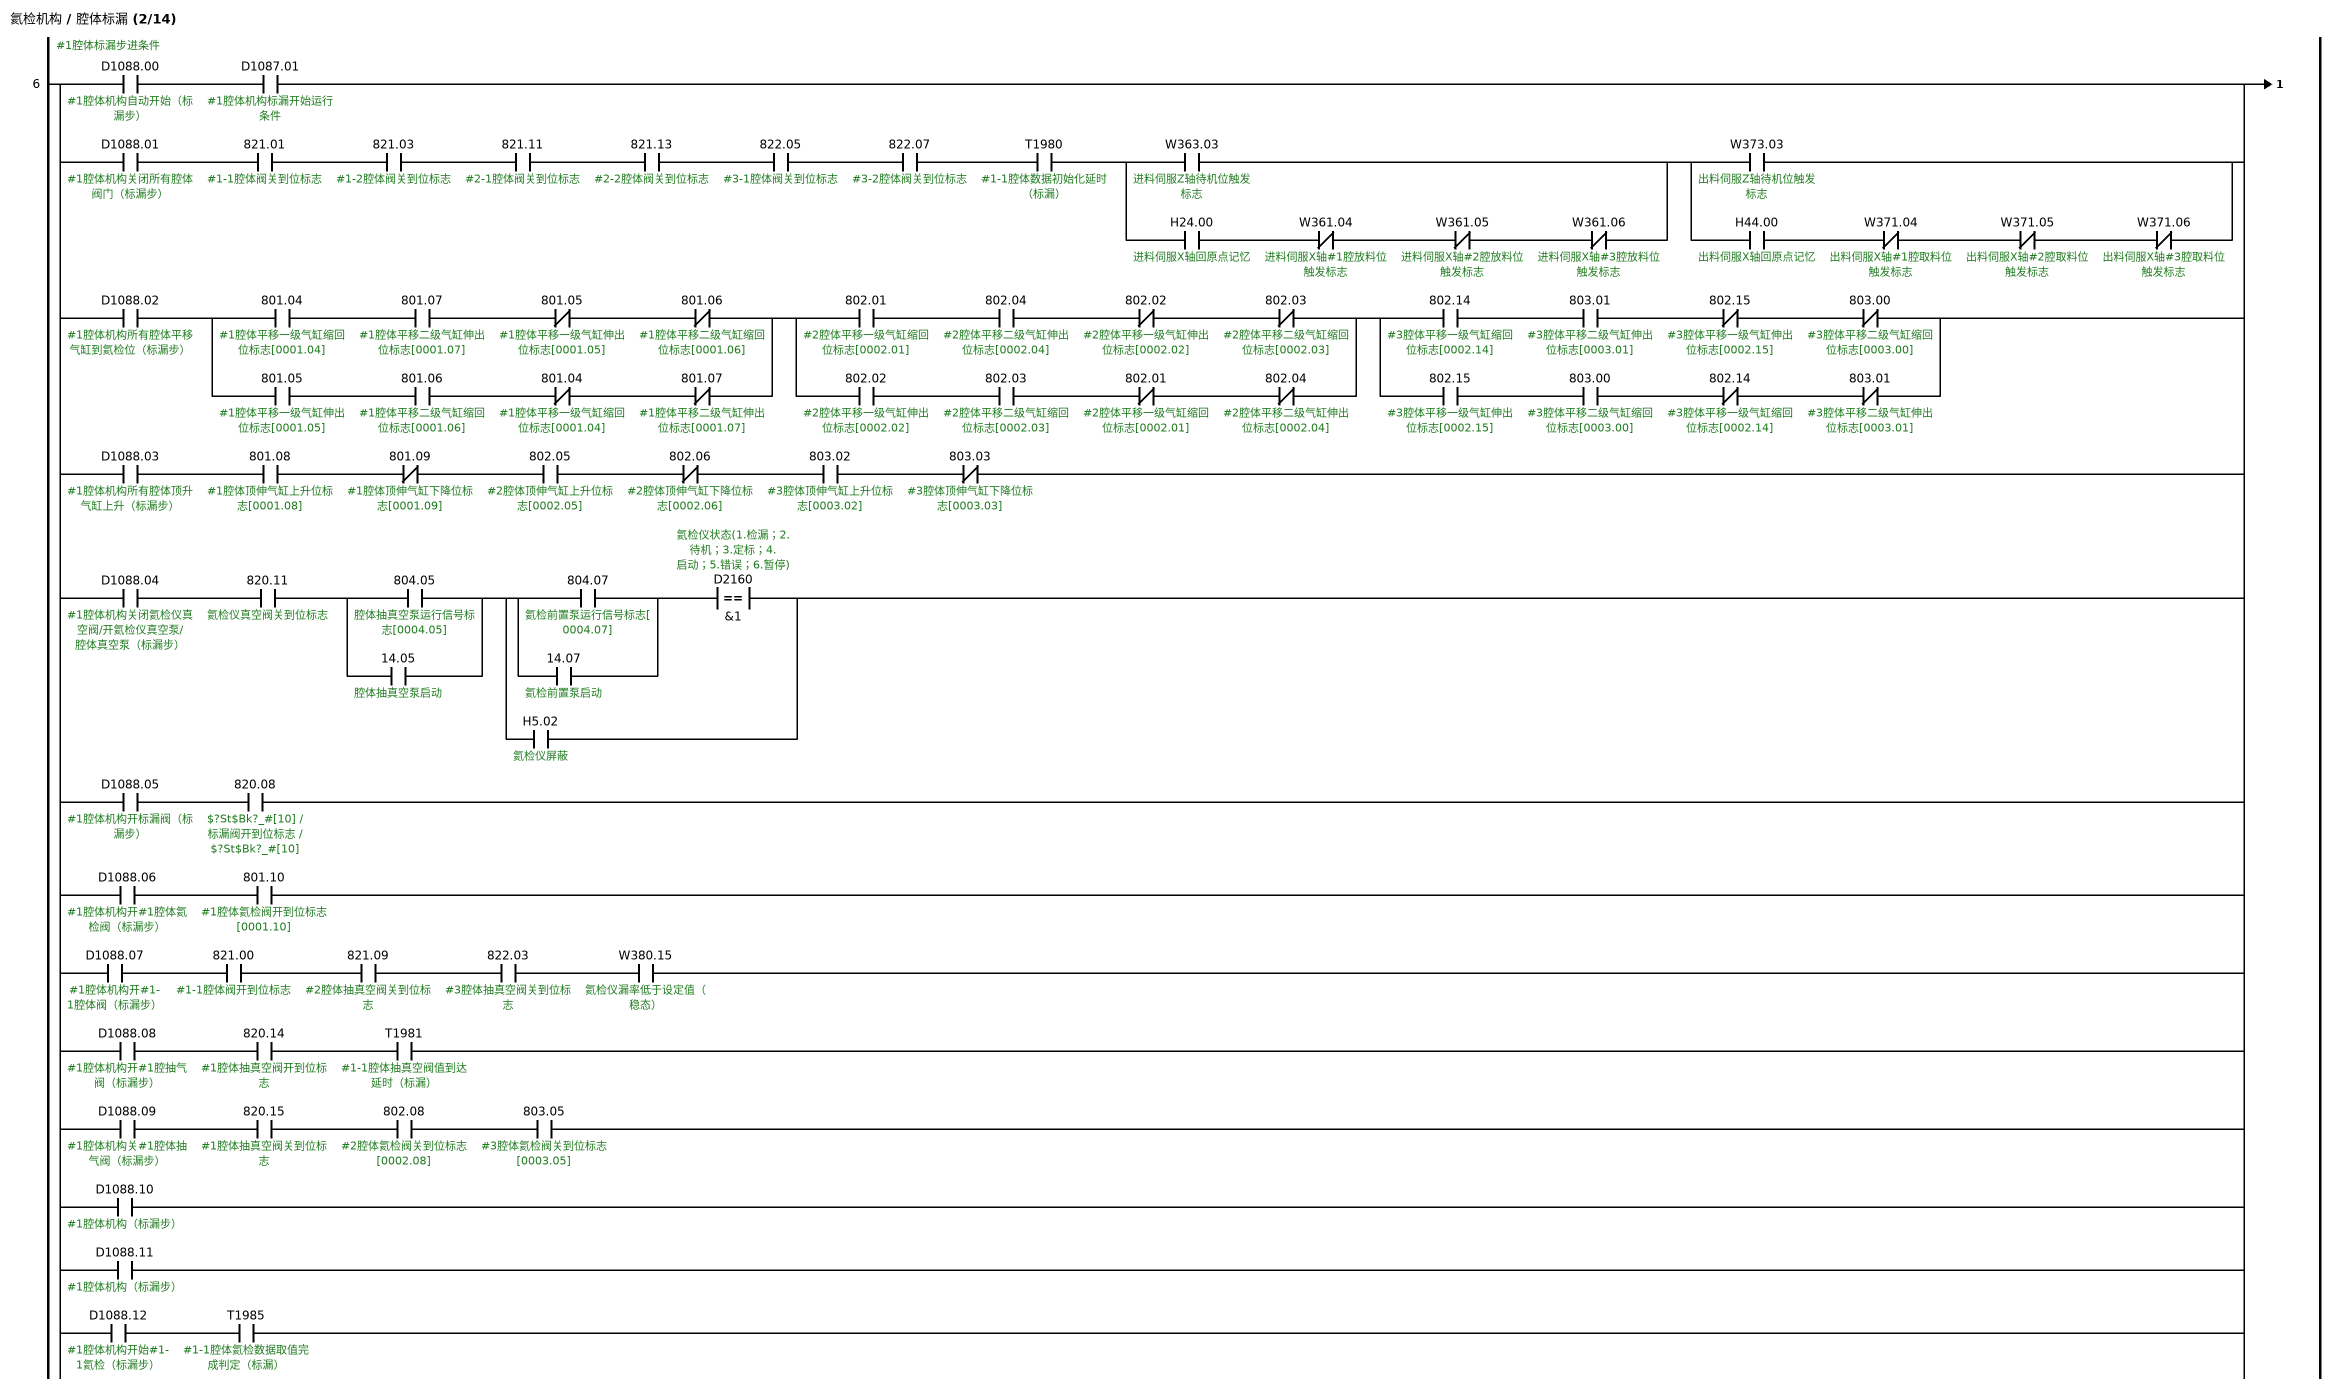

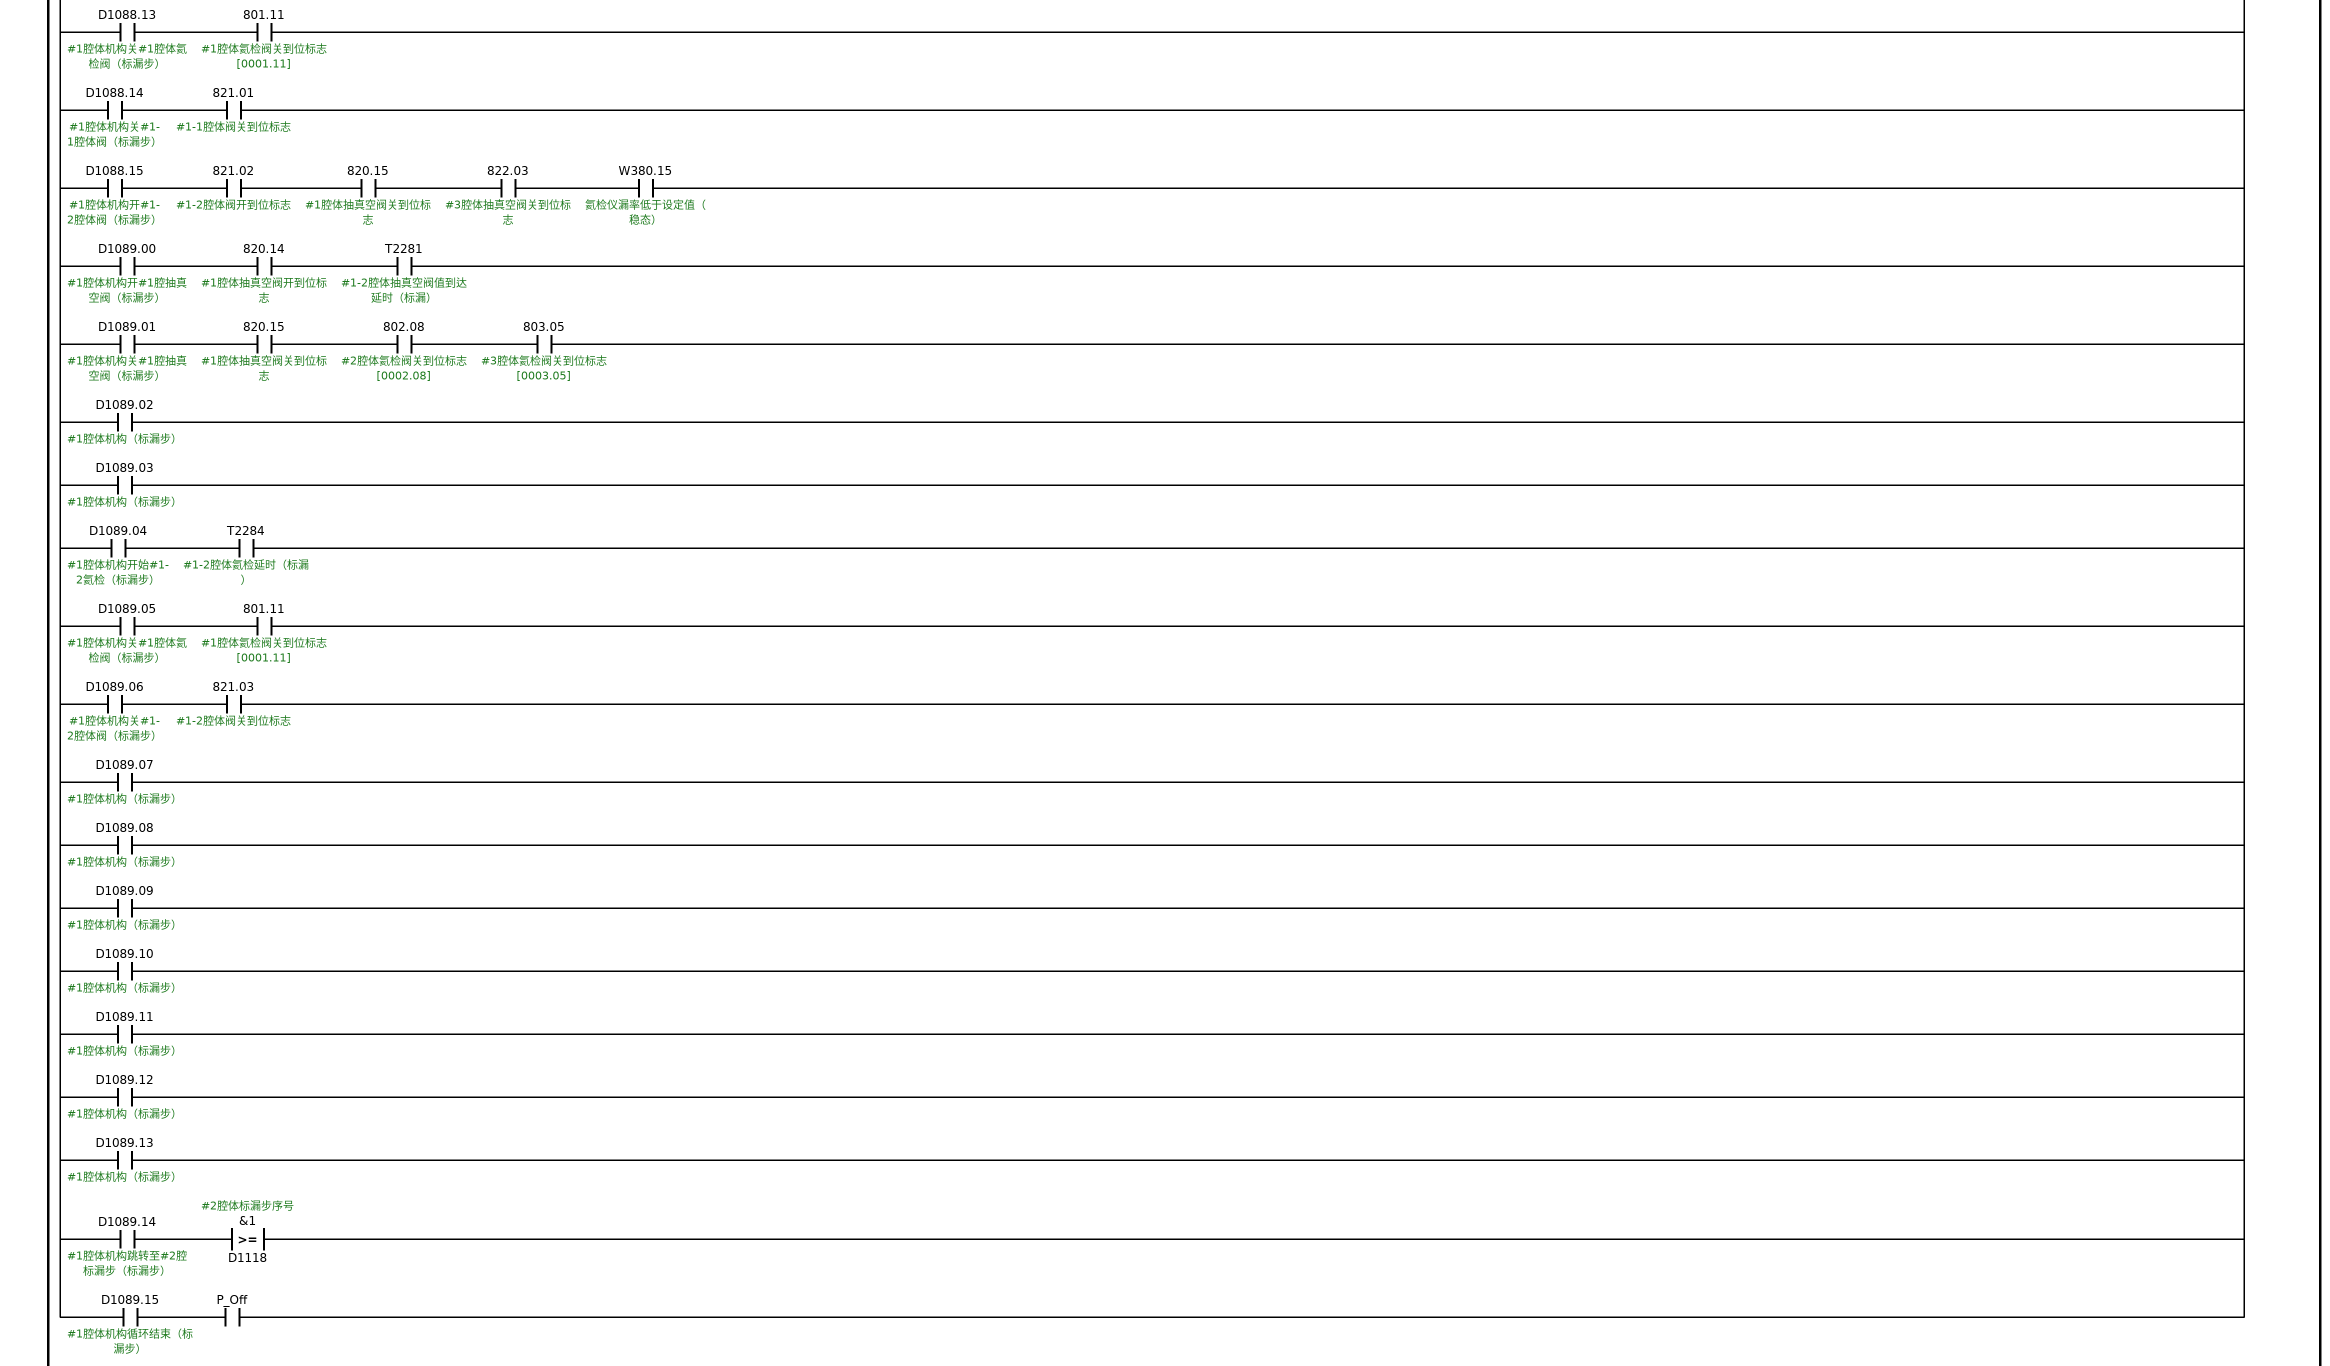

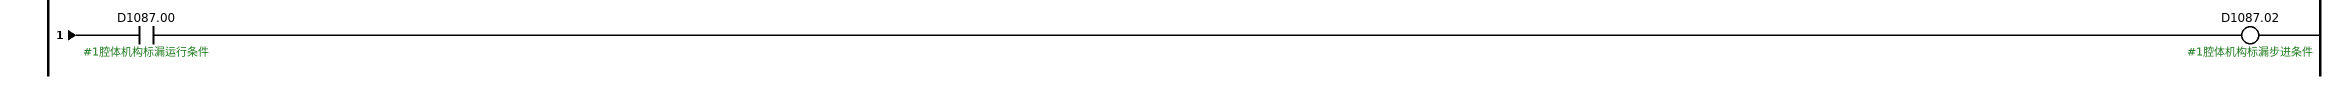
; rung 6: #1腔体标漏步进条件
LD D1088.00  ; #1腔体机构自动开始（标漏步）
AND D1087.01  ; #1腔体机构标漏开始运行条件
LD D1088.01  ; #1腔体机构关闭所有腔体阀门（标漏步）
AND 821.01  ; #1-1腔体阀关到位标志
AND 821.03  ; #1-2腔体阀关到位标志
AND 821.11  ; #2-1腔体阀关到位标志
AND 821.13  ; #2-2腔体阀关到位标志
AND 822.05  ; #3-1腔体阀关到位标志
AND 822.07  ; #3-2腔体阀关到位标志
AND T1980  ; #1-1腔体数据初始化延时（标漏）
LD W363.03  ; 进料伺服Z轴待机位触发标志
LD H24.00  ; 进料伺服X轴回原点记忆
ANDNOT W361.04  ; 进料伺服X轴#1腔放料位触发标志
ANDNOT W361.05  ; 进料伺服X轴#2腔放料位触发标志
ANDNOT W361.06  ; 进料伺服X轴#3腔放料位触发标志
ORLD
ANDLD
LD W373.03  ; 出料伺服Z轴待机位触发标志
LD H44.00  ; 出料伺服X轴回原点记忆
ANDNOT W371.04  ; 出料伺服X轴#1腔取料位触发标志
ANDNOT W371.05  ; 出料伺服X轴#2腔取料位触发标志
ANDNOT W371.06  ; 出料伺服X轴#3腔取料位触发标志
ORLD
ANDLD
ORLD
LD D1088.02  ; #1腔体机构所有腔体平移气缸到氦检位（标漏步）
LD 801.04  ; #1腔体平移一级气缸缩回位标志[0001.04]
AND 801.07  ; #1腔体平移二级气缸伸出位标志[0001.07]
ANDNOT 801.05  ; #1腔体平移一级气缸伸出位标志[0001.05]
ANDNOT 801.06  ; #1腔体平移二级气缸缩回位标志[0001.06]
LD 801.05  ; #1腔体平移一级气缸伸出位标志[0001.05]
AND 801.06  ; #1腔体平移二级气缸缩回位标志[0001.06]
ANDNOT 801.04  ; #1腔体平移一级气缸缩回位标志[0001.04]
ANDNOT 801.07  ; #1腔体平移二级气缸伸出位标志[0001.07]
ORLD
ANDLD
LD 802.01  ; #2腔体平移一级气缸缩回位标志[0002.01]
AND 802.04  ; #2腔体平移二级气缸伸出位标志[0002.04]
ANDNOT 802.02  ; #2腔体平移一级气缸伸出位标志[0002.02]
ANDNOT 802.03  ; #2腔体平移二级气缸缩回位标志[0002.03]
LD 802.02  ; #2腔体平移一级气缸伸出位标志[0002.02]
AND 802.03  ; #2腔体平移二级气缸缩回位标志[0002.03]
ANDNOT 802.01  ; #2腔体平移一级气缸缩回位标志[0002.01]
ANDNOT 802.04  ; #2腔体平移二级气缸伸出位标志[0002.04]
ORLD
ANDLD
LD 802.14  ; #3腔体平移一级气缸缩回位标志[0002.14]
AND 803.01  ; #3腔体平移二级气缸伸出位标志[0003.01]
ANDNOT 802.15  ; #3腔体平移一级气缸伸出位标志[0002.15]
ANDNOT 803.00  ; #3腔体平移二级气缸缩回位标志[0003.00]
LD 802.15  ; #3腔体平移一级气缸伸出位标志[0002.15]
AND 803.00  ; #3腔体平移二级气缸缩回位标志[0003.00]
ANDNOT 802.14  ; #3腔体平移一级气缸缩回位标志[0002.14]
ANDNOT 803.01  ; #3腔体平移二级气缸伸出位标志[0003.01]
ORLD
ANDLD
ORLD
LD D1088.03  ; #1腔体机构所有腔体顶升气缸上升（标漏步）
AND 801.08  ; #1腔体顶伸气缸上升位标志[0001.08]
ANDNOT 801.09  ; #1腔体顶伸气缸下降位标志[0001.09]
AND 802.05  ; #2腔体顶伸气缸上升位标志[0002.05]
ANDNOT 802.06  ; #2腔体顶伸气缸下降位标志[0002.06]
AND 803.02  ; #3腔体顶伸气缸上升位标志[0003.02]
ANDNOT 803.03  ; #3腔体顶伸气缸下降位标志[0003.03]
ORLD
LD D1088.04  ; #1腔体机构关闭氦检仪真空阀/开氦检仪真空泵/腔体真空泵（标漏步）
AND 820.11  ; 氦检仪真空阀关到位标志
LD 804.05  ; 腔体抽真空泵运行信号标志[0004.05]
OR 14.05  ; 腔体抽真空泵启动
ANDLD
LD 804.07  ; 氦检前置泵运行信号标志[0004.07]
OR 14.07  ; 氦检前置泵启动
AND=(300) D2160 &1  ; 氦检仪状态(1.检漏；2.待机；3.定标；4.启动；5.错误；6.暂停)
OR H5.02  ; 氦检仪屏蔽
ANDLD
ORLD
LD D1088.05  ; #1腔体机构开标漏阀（标漏步）
AND 820.08  ; $?St$Bk?_#[10] / 标漏阀开到位标志 / $?St$Bk?_#[10]
ORLD
LD D1088.06  ; #1腔体机构开#1腔体氦检阀（标漏步）
AND 801.10  ; #1腔体氦检阀开到位标志[0001.10]
ORLD
LD D1088.07  ; #1腔体机构开#1-1腔体阀（标漏步）
AND 821.00  ; #1-1腔体阀开到位标志
AND 821.09  ; #2腔体抽真空阀关到位标志
AND 822.03  ; #3腔体抽真空阀关到位标志
AND W380.15  ; 氦检仪漏率低于设定值（稳态）
ORLD
LD D1088.08  ; #1腔体机构开#1腔抽气阀（标漏步）
AND 820.14  ; #1腔体抽真空阀开到位标志
AND T1981  ; #1-1腔体抽真空阀值到达延时（标漏）
ORLD
LD D1088.09  ; #1腔体机构关#1腔体抽气阀（标漏步）
AND 820.15  ; #1腔体抽真空阀关到位标志
AND 802.08  ; #2腔体氦检阀关到位标志[0002.08]
AND 803.05  ; #3腔体氦检阀关到位标志[0003.05]
ORLD
OR D1088.10  ; #1腔体机构（标漏步）
OR D1088.11  ; #1腔体机构（标漏步）
LD D1088.12  ; #1腔体机构开始#1-1氦检（标漏步）
AND T1985  ; #1-1腔体氦检数据取值完成判定（标漏）
ORLD
LD D1088.13  ; #1腔体机构关#1腔体氦检阀（标漏步）
AND 801.11  ; #1腔体氦检阀关到位标志[0001.11]
ORLD
LD D1088.14  ; #1腔体机构关#1-1腔体阀（标漏步）
AND 821.01  ; #1-1腔体阀关到位标志
ORLD
LD D1088.15  ; #1腔体机构开#1-2腔体阀（标漏步）
AND 821.02  ; #1-2腔体阀开到位标志
AND 820.15  ; #1腔体抽真空阀关到位标志
AND 822.03  ; #3腔体抽真空阀关到位标志
AND W380.15  ; 氦检仪漏率低于设定值（稳态）
ORLD
LD D1089.00  ; #1腔体机构开#1腔抽真空阀（标漏步）
AND 820.14  ; #1腔体抽真空阀开到位标志
AND T2281  ; #1-2腔体抽真空阀值到达延时（标漏）
ORLD
LD D1089.01  ; #1腔体机构关#1腔抽真空阀（标漏步）
AND 820.15  ; #1腔体抽真空阀关到位标志
AND 802.08  ; #2腔体氦检阀关到位标志[0002.08]
AND 803.05  ; #3腔体氦检阀关到位标志[0003.05]
ORLD
OR D1089.02  ; #1腔体机构（标漏步）
OR D1089.03  ; #1腔体机构（标漏步）
LD D1089.04  ; #1腔体机构开始#1-2氦检（标漏步）
AND T2284  ; #1-2腔体氦检延时（标漏）
ORLD
LD D1089.05  ; #1腔体机构关#1腔体氦检阀（标漏步）
AND 801.11  ; #1腔体氦检阀关到位标志[0001.11]
ORLD
LD D1089.06  ; #1腔体机构关#1-2腔体阀（标漏步）
AND 821.03  ; #1-2腔体阀关到位标志
ORLD
OR D1089.07  ; #1腔体机构（标漏步）
OR D1089.08  ; #1腔体机构（标漏步）
OR D1089.09  ; #1腔体机构（标漏步）
OR D1089.10  ; #1腔体机构（标漏步）
OR D1089.11  ; #1腔体机构（标漏步）
OR D1089.12  ; #1腔体机构（标漏步）
OR D1089.13  ; #1腔体机构（标漏步）
LD D1089.14  ; #1腔体机构跳转至#2腔标漏步（标漏步）
AND>=L(326) &1 D1118  ; #2腔体标漏步序号
ORLD
LD D1089.15  ; #1腔体机构循环结束（标漏步）
AND P_Off
ORLD
AND D1087.00  ; #1腔体机构标漏运行条件
OUT D1087.02  ; #1腔体机构标漏步进条件

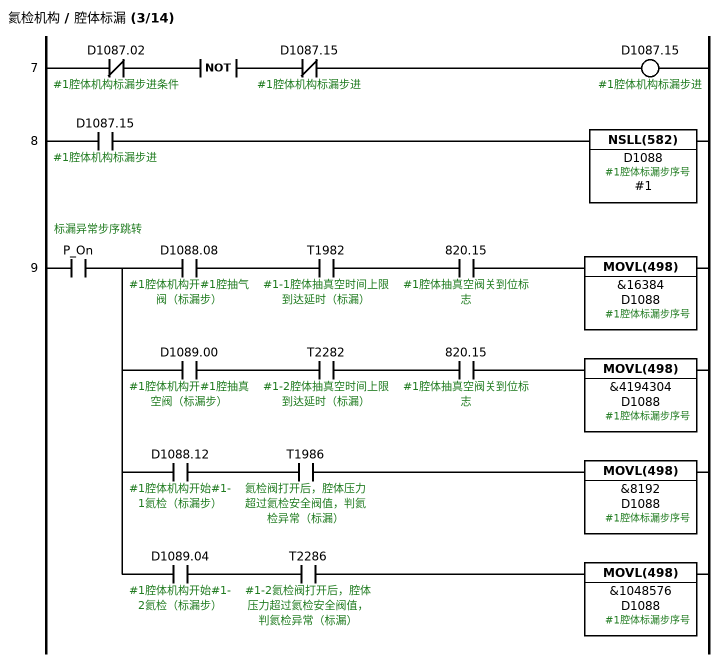
; rung 7
LDNOT D1087.02  ; #1腔体机构标漏步进条件
NOT(520)
ANDNOT D1087.15  ; #1腔体机构标漏步进
OUT D1087.15  ; #1腔体机构标漏步进
; rung 8
LD D1087.15  ; #1腔体机构标漏步进
NSLL(582) D1088 #1  ; #1腔体标漏步序号
; rung 9: 标漏异常步序跳转
LD P_On
OUT TR0
AND D1088.08  ; #1腔体机构开#1腔抽气阀（标漏步）
AND T1982  ; #1-1腔体抽真空时间上限到达延时（标漏）
AND 820.15  ; #1腔体抽真空阀关到位标志
MOVL(498) &16384 D1088  ; #1腔体标漏步序号
LD TR0
AND D1089.00  ; #1腔体机构开#1腔抽真空阀（标漏步）
AND T2282  ; #1-2腔体抽真空时间上限到达延时（标漏）
AND 820.15  ; #1腔体抽真空阀关到位标志
MOVL(498) &4194304 D1088  ; #1腔体标漏步序号
LD TR0
AND D1088.12  ; #1腔体机构开始#1-1氦检（标漏步）
AND T1986  ; 氦检阀打开后，腔体压力超过氦检安全阀值，判氦检异常（标漏）
MOVL(498) &8192 D1088  ; #1腔体标漏步序号
LD TR0
AND D1089.04  ; #1腔体机构开始#1-2氦检（标漏步）
AND T2286  ; #1-2氦检阀打开后，腔体压力超过氦检安全阀值，判氦检异常（标漏）
MOVL(498) &1048576 D1088  ; #1腔体标漏步序号

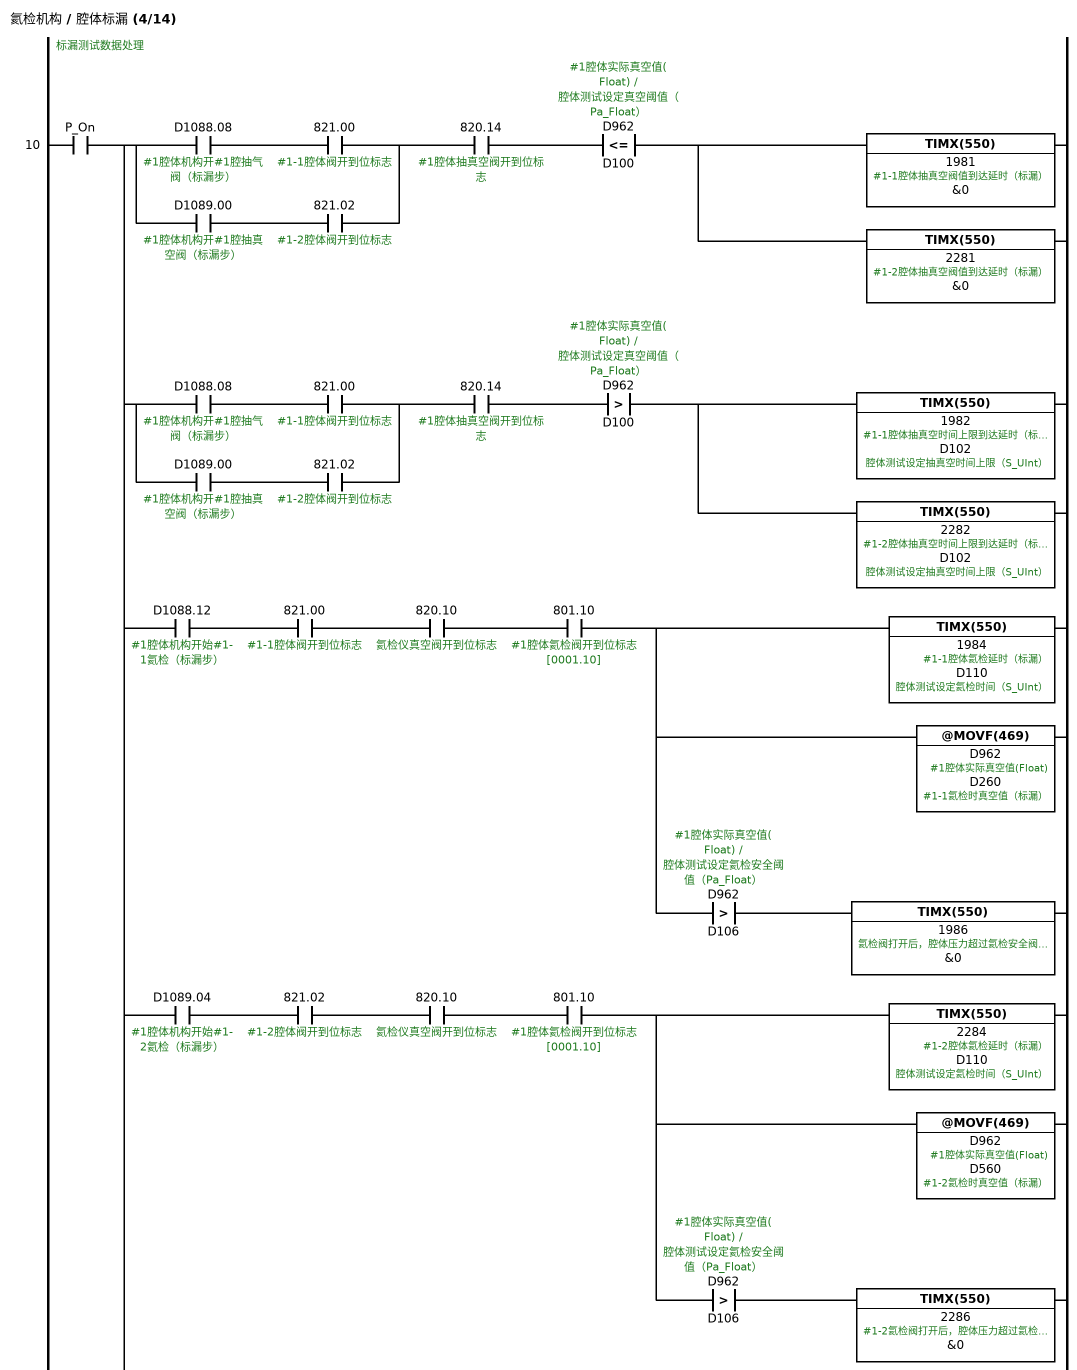

